KUKA KRL program: f1_Kuka_APT209T02S09.SRC

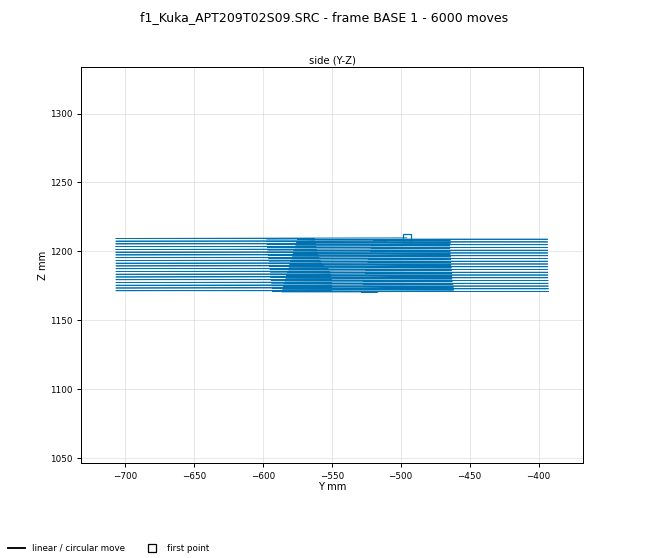
[picture p0: tool path of f1_Kuka_APT209T02S09.SRC in frame BASE 1, 6000 of 6001 moves have a stored position in this frame; points joined in program order, loops and branches not executed]
&ACCESS RVP
&REL 2
&PARAM TEMPLATE = C:\KRC\Roboter\Template\vorgabe
&PARAM EDITMASK = *
DEF f1_Kuka_APT209T02S09()


;FOLD INI;%{PE}%V3.2.0,%MKUKATPBASIS,%CINIT,%VCOMMON,%P
  ;FOLD BAS INI;%{E}%V3.2.0,%MKUKATPBASIS,%CINIT,%VINIT,%P
    GLOBAL INTERRUPT DECL 3 WHEN $STOPMESS==TRUE DO IR_STOPM ( )
    INTERRUPT ON 3
    BAS (#INITMOV,0 )
  ;ENDFOLD (BAS INI)
  ;FOLD USER INI;%{E}%V3.2.0,%MKUKATPUSER,%CINIT,%VINIT,%P
    ;Make your modifications here
  ;ENDFOLD (USER INI)
;ENDFOLD (INI)


;*** Make Null PTP Move
  PTP $pos_act

;*** Auto Load The Correct TOOL Data
  $tool=tool_data[2]

;*** Auto Load The Correct BASE Data
  $base=base_data[1]

  $ADVANCE = 5

;*** Restate Last Velocity
MMPM(30000.0)
SetRPM(8000)
LIN {X 0.139,Y -495.504,Z 1209.880,A 0.000,B 0.000,C 90.000,E1 194.426} C_DIS
LIN {X -0.101,Y -498.909,Z 1209.874,A 0.000,B 0.000,C 90.000,E1 193.244} C_DIS
LIN {X -0.001,Y -505.040,Z 1209.862,A 0.000,B 0.000,C 90.000,E1 191.130} C_DIS
LIN {X 0.236,Y -509.405,Z 1209.854,A 0.000,B 0.000,C 90.000,E1 189.613} C_DIS
LIN {X -0.068,Y -515.059,Z 1209.844,A 0.000,B 0.000,C 90.000,E1 187.871} C_DIS
LIN {X 0.218,Y -518.809,Z 1209.837,A 0.000,B 0.000,C 90.000,E1 186.663} C_DIS
LIN {X 0.043,Y -523.311,Z 1209.829,A 0.000,B 0.000,C 90.000,E1 185.220} C_DIS
LIN {X -0.139,Y -528.677,Z 1209.819,A 0.000,B 0.000,C 90.000,E1 183.498} C_DIS
LIN {X -0.218,Y -533.146,Z 1209.811,A 0.000,B 0.000,C 90.000,E1 182.064} C_DIS
LIN {X -0.220,Y -537.647,Z 1209.803,A 0.000,B 0.000,C 90.000,E1 180.630} C_DIS
LIN {X -0.152,Y -542.076,Z 1209.796,A 0.000,B 0.000,C 90.000,E1 179.198} C_DIS
LIN {X -0.025,Y -545.583,Z 1209.789,A 0.000,B 0.000,C 90.000,E1 178.051} C_DIS
LIN {X 0.254,Y -550.664,Z 1209.780,A 0.000,B 0.000,C 90.000,E1 176.331} C_DIS
LIN {X 0.057,Y -554.716,Z 1209.772,A 0.000,B 0.000,C 90.000,E1 174.951} C_DIS
LIN {X -0.073,Y -558.723,Z 1209.764,A 0.000,B 0.000,C 90.000,E1 173.571} C_DIS
LIN {X 0.229,Y -564.136,Z 1209.754,A 0.000,B 0.000,C 90.000,E1 171.602} C_DIS
LIN {X -0.065,Y -568.767,Z 1209.744,A 0.000,B 0.000,C 90.000,E1 169.982} C_DIS
LIN {X -0.066,Y -573.325,Z 1209.735,A 0.000,B 0.000,C 90.000,E1 168.342} C_DIS
LIN {X 0.038,Y -577.922,Z 1209.726,A 0.000,B 0.000,C 90.000,E1 166.700} C_DIS
LIN {X -0.191,Y -582.656,Z 1209.717,A 0.000,B 0.000,C 90.000,E1 165.102} C_DIS
LIN {X 0.077,Y -588.302,Z 1209.707,A 0.000,B 0.000,C 90.000,E1 163.196} C_DIS
LIN {X 0.217,Y -593.215,Z 1209.698,A 0.000,B 0.000,C 90.000,E1 161.583} C_DIS
LIN {X 0.145,Y -601.075,Z 1209.685,A 0.000,B 0.000,C 90.000,E1 159.209} C_DIS
LIN {X -0.248,Y -607.551,Z 1209.674,A 0.000,B 0.000,C 90.000,E1 157.411} C_DIS
LIN {X 0.351,Y -612.972,Z 1209.666,A 0.000,B 0.000,C 90.000,E1 155.793} C_DIS
LIN {X -0.046,Y -617.299,Z 1209.659,A 0.000,B 0.000,C 90.000,E1 154.537} C_DIS
LIN {X -0.107,Y -621.487,Z 1209.651,A 0.000,B 0.000,C 90.000,E1 153.256} C_DIS
LIN {X -0.107,Y -624.711,Z 1209.646,A 0.000,B 0.000,C 90.000,E1 152.231} C_DIS
LIN {X -0.265,Y -630.161,Z 1209.636,A 0.000,B 0.000,C 90.000,E1 150.461} C_DIS
LIN {X -0.368,Y -633.922,Z 1209.629,A 0.000,B 0.000,C 90.000,E1 149.203} C_DIS
LIN {X 0.090,Y -636.876,Z 1209.623,A 0.000,B 0.000,C 90.000,E1 148.152} C_DIS
LIN {X -0.114,Y -640.335,Z 1209.616,A 0.000,B 0.000,C 90.000,E1 146.914} C_DIS
LIN {X 0.231,Y -642.880,Z 1209.611,A 0.000,B 0.000,C 90.000,E1 145.881} C_DIS
LIN {X 0.127,Y -645.937,Z 1209.604,A 0.000,B 0.000,C 90.000,E1 144.642} C_DIS
LIN {X -0.080,Y -648.713,Z 1209.597,A 0.000,B 0.000,C 90.000,E1 143.417} C_DIS
LIN {X -0.235,Y -651.341,Z 1209.590,A 0.000,B 0.000,C 90.000,E1 142.190} C_DIS
LIN {X 0.060,Y -653.919,Z 1209.583,A 0.000,B 0.000,C 90.000,E1 140.928} C_DIS
LIN {X -0.103,Y -657.497,Z 1209.573,A 0.000,B 0.000,C 90.000,E1 139.218} C_DIS
LIN {X 0.237,Y -661.234,Z 1209.564,A 0.000,B 0.000,C 90.000,E1 137.472} C_DIS
LIN {X -0.311,Y -664.353,Z 1209.556,A 0.000,B 0.000,C 90.000,E1 136.053} C_DIS
LIN {X -0.324,Y -669.340,Z 1209.544,A 0.000,B 0.000,C 90.000,E1 133.866} C_DIS
LIN {X -0.205,Y -673.548,Z 1209.534,A 0.000,B 0.000,C 90.000,E1 132.162} C_DIS
LIN {X -0.016,Y -677.073,Z 1209.526,A 0.000,B 0.000,C 90.000,E1 130.701} C_DIS
LIN {X 0.170,Y -679.469,Z 1209.521,A 0.000,B 0.000,C 90.000,E1 129.725} C_DIS
LIN {X 0.021,Y -683.002,Z 1209.513,A 0.000,B 0.000,C 90.000,E1 128.302} C_DIS
LIN {X -0.325,Y -687.178,Z 1209.504,A 0.000,B 0.000,C 90.000,E1 126.664} C_DIS
LIN {X -0.075,Y -688.967,Z 1209.500,A 0.000,B 0.000,C 90.000,E1 125.931} C_DIS
LIN {X 0.231,Y -692.270,Z 1209.492,A 0.000,B 0.000,C 90.000,E1 124.485} C_DIS
LIN {X -0.226,Y -694.400,Z 1209.486,A 0.000,B 0.000,C 90.000,E1 123.579} C_DIS
LIN {X -0.426,Y -696.993,Z 1209.480,A 0.000,B 0.000,C 90.000,E1 122.418} C_DIS
LIN {X 0.093,Y -698.481,Z 1209.476,A 0.000,B 0.000,C 90.000,E1 121.671} C_DIS
LIN {X -0.055,Y -700.752,Z 1209.469,A 0.000,B 0.000,C 90.000,E1 120.512} C_DIS
LIN {X 0.075,Y -702.947,Z 1209.463,A 0.000,B 0.000,C 90.000,E1 119.333} C_DIS
LIN {X -0.041,Y -704.508,Z 1209.458,A 0.000,B 0.000,C 90.000,E1 118.409} C_DIS
LIN {X -0.425,Y -705.192,Z 1209.455,A 0.000,B 0.000,C 90.000,E1 117.975} C_DIS
LIN {X -0.181,Y -705.879,Z 1209.451,A 0.000,B 0.000,C 90.000,E1 117.257} C_DIS
LIN {X 0.043,Y -706.510,Z 1209.446,A 0.000,B 0.000,C 90.000,E1 116.309} C_DIS
LIN {X 0.292,Y -706.772,Z 1209.442,A 0.000,B 0.000,C 90.000,E1 115.591} C_DIS
LIN {X -0.060,Y -706.742,Z 1209.440,A 0.000,B 0.000,C 90.000,E1 115.155} C_DIS
LIN {X -0.115,Y -706.152,Z 1209.436,A 0.000,B 0.000,C 90.000,E1 114.463} C_DIS
LIN {X -0.177,Y -705.283,Z 1209.433,A 0.000,B 0.000,C 90.000,E1 114.003} C_DIS
LIN {X -0.175,Y -704.420,Z 1209.432,A 0.000,B 0.000,C 90.000,E1 113.770} C_DIS
LIN {X 0.391,Y -702.162,Z 1209.429,A 0.000,B 0.000,C 90.000,E1 113.259} C_DIS
LIN {X -0.391,Y -701.273,Z 1209.429,A 0.000,B 0.000,C 90.000,E1 113.206} C_DIS
LIN {X -0.049,Y -698.541,Z 1209.427,A 0.000,B 0.000,C 90.000,E1 112.950} C_DIS
LIN {X -0.168,Y -694.330,Z 1209.426,A 0.000,B 0.000,C 90.000,E1 112.642} C_DIS
LIN {X 0.180,Y -692.034,Z 1209.425,A 0.000,B 0.000,C 90.000,E1 112.514} C_DIS
LIN {X -0.156,Y -687.353,Z 1209.424,A 0.000,B 0.000,C 90.000,E1 112.386} C_DIS
LIN {X -0.201,Y -685.168,Z 1209.424,A 0.000,B 0.000,C 90.000,E1 112.333} C_DIS
LIN {X 0.019,Y -676.728,Z 1209.424,A 0.000,B 0.000,C 90.000,E1 112.280} C_DIS
LIN {X -0.017,Y -610.154,Z 1209.424,A 0.000,B 0.000,C 90.000,E1 112.280} C_DIS
LIN {X -0.099,Y -607.762,Z 1209.423,A 0.000,B 0.000,C 90.000,E1 112.153} C_DIS
LIN {X 0.206,Y -603.602,Z 1209.422,A 0.000,B 0.000,C 90.000,E1 111.844} C_DIS
LIN {X -0.326,Y -599.261,Z 1209.420,A 0.000,B 0.000,C 90.000,E1 111.535} C_DIS
LIN {X -0.044,Y -596.935,Z 1209.418,A 0.000,B 0.000,C 90.000,E1 111.280} C_DIS
LIN {X -0.020,Y -595.513,Z 1209.418,A 0.000,B 0.000,C 90.000,E1 111.153} C_DIS
LIN {X -0.208,Y -594.337,Z 1209.417,A 0.000,B 0.000,C 90.000,E1 111.046} C_DIS
LIN {X -0.049,Y -592.336,Z 1209.416,A 0.000,B 0.000,C 90.000,E1 110.791} C_DIS
LIN {X -0.092,Y -592.311,Z 1209.416,A 0.000,B 0.000,C 90.000,E1 110.791} C_DIS
LIN {X 0.096,Y -591.736,Z 1209.414,A 0.000,B 0.000,C 90.000,E1 110.482} C_DIS
LIN {X -0.232,Y -592.138,Z 1209.412,A 0.000,B 0.000,C 90.000,E1 110.248} C_DIS
LIN {X -0.086,Y -596.332,Z 1209.405,A 0.000,B 0.000,C 90.000,E1 108.906} C_DIS
LIN {X -0.199,Y -597.165,Z 1209.404,A 0.000,B 0.000,C 90.000,E1 108.652} C_DIS
LIN {X -0.167,Y -602.046,Z 1209.393,A 0.000,B 0.000,C 90.000,E1 106.804} C_DIS
LIN {X 0.023,Y -603.299,Z 1209.390,A 0.000,B 0.000,C 90.000,E1 106.260} C_DIS
LIN {X 0.260,Y -605.497,Z 1209.385,A 0.000,B 0.000,C 90.000,E1 105.190} C_DIS
LIN {X -0.065,Y -606.611,Z 1209.379,A 0.000,B 0.000,C 90.000,E1 104.175} C_DIS
LIN {X -0.266,Y -606.970,Z 1209.374,A 0.000,B 0.000,C 90.000,E1 103.411} C_DIS
LIN {X -0.199,Y -606.754,Z 1209.371,A 0.000,B 0.000,C 90.000,E1 102.883} C_DIS
LIN {X 0.129,Y -606.556,Z 1209.370,A 0.000,B 0.000,C 90.000,E1 102.591} C_DIS
LIN {X 0.195,Y -605.757,Z 1209.367,A 0.000,B 0.000,C 90.000,E1 102.063} C_DIS
LIN {X 0.255,Y -604.578,Z 1209.364,A 0.000,B 0.000,C 90.000,E1 101.535} C_DIS
LIN {X 0.305,Y -602.971,Z 1209.361,A 0.000,B 0.000,C 90.000,E1 101.007} C_DIS
LIN {X -0.084,Y -601.975,Z 1209.360,A 0.000,B 0.000,C 90.000,E1 100.782} C_DIS
LIN {X -0.048,Y -599.580,Z 1209.357,A 0.000,B 0.000,C 90.000,E1 100.254} C_DIS
LIN {X -0.035,Y -596.738,Z 1209.354,A 0.000,B 0.000,C 90.000,E1 99.726} C_DIS
LIN {X 0.055,Y -594.326,Z 1209.352,A 0.000,B 0.000,C 90.000,E1 99.321} C_DIS
LIN {X -0.180,Y -589.543,Z 1209.348,A 0.000,B 0.000,C 90.000,E1 98.681} C_DIS
LIN {X 0.248,Y -585.132,Z 1209.345,A 0.000,B 0.000,C 90.000,E1 98.106} C_DIS
LIN {X -0.230,Y -581.136,Z 1209.343,A 0.000,B 0.000,C 90.000,E1 97.757} C_DIS
LIN {X 0.097,Y -578.320,Z 1209.342,A 0.000,B 0.000,C 90.000,E1 97.473} C_DIS
LIN {X 0.147,Y -572.423,Z 1209.339,A 0.000,B 0.000,C 90.000,E1 97.004} C_DIS
LIN {X -0.278,Y -569.383,Z 1209.338,A 0.000,B 0.000,C 90.000,E1 96.834} C_DIS
LIN {X -0.203,Y -568.061,Z 1209.337,A 0.000,B 0.000,C 90.000,E1 96.720} C_DIS
LIN {X -0.262,Y -564.683,Z 1209.335,A 0.000,B 0.000,C 90.000,E1 96.372} C_DIS
LIN {X 0.221,Y -564.184,Z 1209.335,A 0.000,B 0.000,C 90.000,E1 96.258} C_DIS
LIN {X 0.042,Y -563.353,Z 1209.334,A 0.000,B 0.000,C 90.000,E1 96.087} C_DIS
LIN {X 0.089,Y -563.274,Z 1209.333,A 0.000,B 0.000,C 90.000,E1 95.910} C_DIS
LIN {X 0.180,Y -562.863,Z 1209.331,A 0.000,B 0.000,C 90.000,E1 95.625} C_DIS
LIN {X -0.049,Y -562.866,Z 1209.327,A 0.000,B 0.000,C 90.000,E1 94.821} C_DIS
LIN {X -0.096,Y -564.202,Z 1209.313,A 0.000,B 0.000,C 90.000,E1 92.350} C_DIS
LIN {X -0.212,Y -565.047,Z 1209.307,A 0.000,B 0.000,C 90.000,E1 91.260} C_DIS
LIN {X -0.217,Y -566.044,Z 1209.299,A 0.000,B 0.000,C 90.000,E1 89.885} C_DIS
LIN {X 0.166,Y -567.706,Z 1209.287,A 0.000,B 0.000,C 90.000,E1 87.650} C_DIS
LIN {X -0.069,Y -569.116,Z 1209.276,A 0.000,B 0.000,C 90.000,E1 85.755} C_DIS
LIN {X 0.169,Y -570.459,Z 1209.267,A 0.000,B 0.000,C 90.000,E1 84.090} C_DIS
LIN {X -0.015,Y -571.749,Z 1209.258,A 0.000,B 0.000,C 90.000,E1 82.470} C_DIS
LIN {X 0.209,Y -572.803,Z 1209.251,A 0.000,B 0.000,C 90.000,E1 81.084} C_DIS
LIN {X 0.169,Y -573.886,Z 1209.242,A 0.000,B 0.000,C 90.000,E1 79.454} C_DIS
LIN {X 0.144,Y -574.948,Z 1209.233,A 0.000,B 0.000,C 90.000,E1 77.825} C_DIS
LIN {X -0.177,Y -575.786,Z 1209.223,A 0.000,B 0.000,C 90.000,E1 76.228} C_DIS
LIN {X -0.266,Y -576.758,Z 1209.213,A 0.000,B 0.000,C 90.000,E1 74.338} C_DIS
LIN {X 0.161,Y -577.655,Z 1209.204,A 0.000,B 0.000,C 90.000,E1 72.670} C_DIS
LIN {X 0.062,Y -578.729,Z 1209.193,A 0.000,B 0.000,C 90.000,E1 70.786} C_DIS
LIN {X -0.004,Y -580.016,Z 1209.183,A 0.000,B 0.000,C 90.000,E1 68.901} C_DIS
LIN {X 0.155,Y -581.553,Z 1209.172,A 0.000,B 0.000,C 90.000,E1 66.997} C_DIS
LIN {X -0.123,Y -583.097,Z 1209.163,A 0.000,B 0.000,C 90.000,E1 65.409} C_DIS
LIN {X -0.079,Y -585.043,Z 1209.151,A 0.000,B 0.000,C 90.000,E1 63.256} C_DIS
LIN {X -0.014,Y -586.685,Z 1209.142,A 0.000,B 0.000,C 90.000,E1 61.641} C_DIS
LIN {X -0.144,Y -588.289,Z 1209.134,A 0.000,B 0.000,C 90.000,E1 60.049} C_DIS
LIN {X 0.196,Y -589.370,Z 1209.128,A 0.000,B 0.000,C 90.000,E1 58.948} C_DIS
LIN {X -0.079,Y -590.733,Z 1209.119,A 0.000,B 0.000,C 90.000,E1 57.375} C_DIS
LIN {X 0.171,Y -591.978,Z 1209.110,A 0.000,B 0.000,C 90.000,E1 55.754} C_DIS
LIN {X -0.203,Y -593.254,Z 1209.101,A 0.000,B 0.000,C 90.000,E1 54.196} C_DIS
LIN {X 0.283,Y -594.420,Z 1209.092,A 0.000,B 0.000,C 90.000,E1 52.557} C_DIS
LIN {X -0.108,Y -594.844,Z 1209.089,A 0.000,B 0.000,C 90.000,E1 52.065} C_DIS
LIN {X 0.068,Y -596.010,Z 1209.079,A 0.000,B 0.000,C 90.000,E1 50.194} C_DIS
LIN {X 0.058,Y -596.520,Z 1209.073,A 0.000,B 0.000,C 90.000,E1 49.138} C_DIS
LIN {X 0.049,Y -597.057,Z 1209.064,A 0.000,B 0.000,C 90.000,E1 47.553} C_DIS
LIN {X 0.012,Y -597.327,Z 1209.058,A 0.000,B 0.000,C 90.000,E1 46.500} C_DIS
LIN {X 0.197,Y -597.520,Z 1209.051,A 0.000,B 0.000,C 90.000,E1 45.162} C_DIS
LIN {X -0.047,Y -597.259,Z 1209.044,A 0.000,B 0.000,C 90.000,E1 43.866} C_DIS
LIN {X -0.086,Y -596.897,Z 1209.038,A 0.000,B 0.000,C 90.000,E1 42.813} C_DIS
LIN {X -0.098,Y -596.277,Z 1209.032,A 0.000,B 0.000,C 90.000,E1 41.757} C_DIS
LIN {X 0.119,Y -595.801,Z 1209.028,A 0.000,B 0.000,C 90.000,E1 40.943} C_DIS
LIN {X -0.130,Y -594.866,Z 1209.020,A 0.000,B 0.000,C 90.000,E1 39.644} C_DIS
LIN {X 0.075,Y -594.188,Z 1209.016,A 0.000,B 0.000,C 90.000,E1 38.830} C_DIS
LIN {X 0.271,Y -593.372,Z 1209.011,A 0.000,B 0.000,C 90.000,E1 38.016} C_DIS
LIN {X -0.162,Y -592.237,Z 1209.005,A 0.000,B 0.000,C 90.000,E1 36.996} C_DIS
LIN {X 0.069,Y -590.336,Z 1208.998,A 0.000,B 0.000,C 90.000,E1 35.644} C_DIS
LIN {X -0.274,Y -588.357,Z 1208.992,A 0.000,B 0.000,C 90.000,E1 34.612} C_DIS
LIN {X -0.014,Y -586.602,Z 1208.988,A 0.000,B 0.000,C 90.000,E1 33.785} C_DIS
LIN {X 0.225,Y -584.637,Z 1208.983,A 0.000,B 0.000,C 90.000,E1 32.959} C_DIS
LIN {X -0.363,Y -582.233,Z 1208.979,A 0.000,B 0.000,C 90.000,E1 32.212} C_DIS
LIN {X -0.175,Y -579.536,Z 1208.974,A 0.000,B 0.000,C 90.000,E1 31.386} C_DIS
LIN {X 0.326,Y -577.503,Z 1208.971,A 0.000,B 0.000,C 90.000,E1 30.797} C_DIS
LIN {X 0.161,Y -574.088,Z 1208.967,A 0.000,B 0.000,C 90.000,E1 30.001} C_DIS
LIN {X -0.041,Y -570.260,Z 1208.962,A 0.000,B 0.000,C 90.000,E1 29.205} C_DIS
LIN {X 0.298,Y -566.674,Z 1208.958,A 0.000,B 0.000,C 90.000,E1 28.487} C_DIS
LIN {X -0.066,Y -563.567,Z 1208.955,A 0.000,B 0.000,C 90.000,E1 27.975} C_DIS
LIN {X 0.212,Y -559.450,Z 1208.952,A 0.000,B 0.000,C 90.000,E1 27.257} C_DIS
LIN {X 0.090,Y -554.201,Z 1208.947,A 0.000,B 0.000,C 90.000,E1 26.437} C_DIS
LIN {X 0.157,Y -548.224,Z 1208.942,A 0.000,B 0.000,C 90.000,E1 25.591} C_DIS
LIN {X 0.045,Y -542.810,Z 1208.938,A 0.000,B 0.000,C 90.000,E1 24.899} C_DIS
LIN {X -0.110,Y -537.075,Z 1208.934,A 0.000,B 0.000,C 90.000,E1 24.207} C_DIS
LIN {X 0.042,Y -529.607,Z 1208.930,A 0.000,B 0.000,C 90.000,E1 23.334} C_DIS
LIN {X -0.095,Y -523.144,Z 1208.926,A 0.000,B 0.000,C 90.000,E1 22.642} C_DIS
LIN {X -0.038,Y -512.535,Z 1208.920,A 0.000,B 0.000,C 90.000,E1 21.535} C_DIS
LIN {X 0.089,Y -502.840,Z 1208.914,A 0.000,B 0.000,C 90.000,E1 20.556} C_DIS
LIN {X 0.092,Y -493.072,Z 1208.909,A 0.000,B 0.000,C 90.000,E1 19.631} C_DIS
LIN {X -0.078,Y -484.282,Z 1208.905,A 0.000,B 0.000,C 90.000,E1 18.852} C_DIS
LIN {X -0.191,Y -473.999,Z 1208.900,A 0.000,B 0.000,C 90.000,E1 17.946} C_DIS
LIN {X -0.210,Y -459.021,Z 1208.892,A 0.000,B 0.000,C 90.000,E1 16.622} C_DIS
LIN {X 0.052,Y -437.190,Z 1208.881,A 0.000,B 0.000,C 90.000,E1 14.537} C_DIS
LIN {X 0.049,Y -421.688,Z 1208.872,A 0.000,B 0.000,C 90.000,E1 12.939} C_DIS
LIN {X 0.085,Y -404.925,Z 1208.861,A 0.000,B 0.000,C 90.000,E1 11.007} C_DIS
LIN {X 0.068,Y -397.362,Z 1208.856,A 0.000,B 0.000,C 90.000,E1 10.018} C_DIS
LIN {X 0.048,Y -395.305,Z 1208.854,A 0.000,B 0.000,C 90.000,E1 9.670} C_DIS
LIN {X -0.151,Y -393.958,Z 1208.852,A 0.000,B 0.000,C 90.000,E1 9.434} C_DIS
LIN {X -0.107,Y -393.353,Z 1208.851,A 0.000,B 0.000,C 90.000,E1 9.151} C_DIS
LIN {X -0.144,Y -393.341,Z 1208.851,A 0.000,B 0.000,C 90.000,E1 9.151} C_DIS
LIN {X -0.068,Y -393.829,Z 1208.849,A 0.000,B 0.000,C 90.000,E1 8.803} C_DIS
LIN {X -0.142,Y -396.754,Z 1208.845,A 0.000,B 0.000,C 90.000,E1 8.106} C_DIS
LIN {X -0.187,Y -397.947,Z 1208.844,A 0.000,B 0.000,C 90.000,E1 7.936} C_DIS
LIN {X -0.212,Y -400.655,Z 1208.842,A 0.000,B 0.000,C 90.000,E1 7.587} C_DIS
LIN {X 0.204,Y -402.237,Z 1208.841,A 0.000,B 0.000,C 90.000,E1 7.352} C_DIS
LIN {X 0.215,Y -407.342,Z 1208.839,A 0.000,B 0.000,C 90.000,E1 6.891} C_DIS
LIN {X 0.092,Y -426.083,Z 1208.830,A 0.000,B 0.000,C 90.000,E1 5.454} C_DIS
LIN {X 0.154,Y -438.832,Z 1208.825,A 0.000,B 0.000,C 90.000,E1 4.473} C_DIS
LIN {X 0.215,Y -454.780,Z 1208.818,A 0.000,B 0.000,C 90.000,E1 3.269} C_DIS
LIN {X 0.037,Y -464.247,Z 1208.814,A 0.000,B 0.000,C 90.000,E1 2.579} C_DIS
LIN {X -0.223,Y -473.438,Z 1208.810,A 0.000,B 0.000,C 90.000,E1 1.892} C_DIS
LIN {X 0.079,Y -479.294,Z 1208.808,A 0.000,B 0.000,C 90.000,E1 1.375} C_DIS
LIN {X 0.100,Y -485.204,Z 1208.805,A 0.000,B 0.000,C 90.000,E1 0.859} C_DIS
LIN {X -0.057,Y -490.896,Z 1208.802,A 0.000,B 0.000,C 90.000,E1 0.344} C_DIS
LIN {X -0.023,Y -497.632,Z 1208.798,A 0.000,B 0.000,C 90.000,E1 359.656} C_DIS
LIN {X -0.115,Y -505.401,Z 1208.793,A 0.000,B 0.000,C 90.000,E1 358.797} C_DIS
LIN {X -0.060,Y -511.385,Z 1208.789,A 0.000,B 0.000,C 90.000,E1 358.051} C_DIS
LIN {X -0.010,Y -517.010,Z 1208.785,A 0.000,B 0.000,C 90.000,E1 357.306} C_DIS
LIN {X -0.117,Y -521.216,Z 1208.782,A 0.000,B 0.000,C 90.000,E1 356.731} C_DIS
LIN {X 0.013,Y -526.004,Z 1208.778,A 0.000,B 0.000,C 90.000,E1 355.988} C_DIS
LIN {X 0.221,Y -530.323,Z 1208.774,A 0.000,B 0.000,C 90.000,E1 355.241} C_DIS
LIN {X 0.215,Y -533.527,Z 1208.771,A 0.000,B 0.000,C 90.000,E1 354.666} C_DIS
LIN {X 0.233,Y -536.478,Z 1208.767,A 0.000,B 0.000,C 90.000,E1 354.090} C_DIS
LIN {X -0.206,Y -540.361,Z 1208.763,A 0.000,B 0.000,C 90.000,E1 353.280} C_DIS
LIN {X 0.131,Y -543.384,Z 1208.759,A 0.000,B 0.000,C 90.000,E1 352.534} C_DIS
LIN {X -0.245,Y -546.623,Z 1208.754,A 0.000,B 0.000,C 90.000,E1 351.724} C_DIS
LIN {X 0.040,Y -549.539,Z 1208.749,A 0.000,B 0.000,C 90.000,E1 350.849} C_DIS
LIN {X -0.157,Y -552.960,Z 1208.743,A 0.000,B 0.000,C 90.000,E1 349.746} C_DIS
LIN {X -0.207,Y -556.077,Z 1208.737,A 0.000,B 0.000,C 90.000,E1 348.634} C_DIS
LIN {X -0.208,Y -558.908,Z 1208.731,A 0.000,B 0.000,C 90.000,E1 347.521} C_DIS
LIN {X 0.223,Y -560.866,Z 1208.726,A 0.000,B 0.000,C 90.000,E1 346.645} C_DIS
LIN {X -0.129,Y -563.293,Z 1208.720,A 0.000,B 0.000,C 90.000,E1 345.574} C_DIS
LIN {X 0.264,Y -566.109,Z 1208.712,A 0.000,B 0.000,C 90.000,E1 344.157} C_DIS
LIN {X -0.018,Y -568.156,Z 1208.706,A 0.000,B 0.000,C 90.000,E1 343.087} C_DIS
LIN {X -0.107,Y -570.038,Z 1208.700,A 0.000,B 0.000,C 90.000,E1 342.000} C_DIS
LIN {X 0.208,Y -571.336,Z 1208.695,A 0.000,B 0.000,C 90.000,E1 341.148} C_DIS
LIN {X 0.168,Y -572.775,Z 1208.689,A 0.000,B 0.000,C 90.000,E1 340.061} C_DIS
LIN {X -0.023,Y -573.704,Z 1208.685,A 0.000,B 0.000,C 90.000,E1 339.263} C_DIS
LIN {X 0.165,Y -574.623,Z 1208.679,A 0.000,B 0.000,C 90.000,E1 338.156} C_DIS
LIN {X -0.009,Y -574.953,Z 1208.674,A 0.000,B 0.000,C 90.000,E1 337.358} C_DIS
LIN {X 0.043,Y -575.052,Z 1208.670,A 0.000,B 0.000,C 90.000,E1 336.538} C_DIS
LIN {X 0.022,Y -575.001,Z 1208.667,A 0.000,B 0.000,C 90.000,E1 335.997} C_DIS
LIN {X -0.084,Y -574.305,Z 1208.661,A 0.000,B 0.000,C 90.000,E1 334.921} C_DIS
LIN {X 0.119,Y -573.741,Z 1208.658,A 0.000,B 0.000,C 90.000,E1 334.357} C_DIS
LIN {X -0.106,Y -572.527,Z 1208.653,A 0.000,B 0.000,C 90.000,E1 333.563} C_DIS
LIN {X -0.080,Y -570.852,Z 1208.649,A 0.000,B 0.000,C 90.000,E1 332.743} C_DIS
LIN {X 0.186,Y -568.925,Z 1208.644,A 0.000,B 0.000,C 90.000,E1 331.897} C_DIS
LIN {X -0.067,Y -566.664,Z 1208.639,A 0.000,B 0.000,C 90.000,E1 331.101} C_DIS
LIN {X 0.064,Y -564.846,Z 1208.636,A 0.000,B 0.000,C 90.000,E1 330.539} C_DIS
LIN {X -0.036,Y -562.668,Z 1208.633,A 0.000,B 0.000,C 90.000,E1 329.999} C_DIS
LIN {X -0.046,Y -560.751,Z 1208.631,A 0.000,B 0.000,C 90.000,E1 329.587} C_DIS
LIN {X 0.310,Y -557.934,Z 1208.628,A 0.000,B 0.000,C 90.000,E1 328.997} C_DIS
LIN {X 0.053,Y -553.811,Z 1208.624,A 0.000,B 0.000,C 90.000,E1 328.329} C_DIS
LIN {X -0.240,Y -549.077,Z 1208.620,A 0.000,B 0.000,C 90.000,E1 327.661} C_DIS
LIN {X 0.181,Y -544.010,Z 1208.616,A 0.000,B 0.000,C 90.000,E1 326.914} C_DIS
LIN {X -0.061,Y -539.580,Z 1208.613,A 0.000,B 0.000,C 90.000,E1 326.373} C_DIS
LIN {X -0.096,Y -531.519,Z 1208.608,A 0.000,B 0.000,C 90.000,E1 325.388} C_DIS
LIN {X -0.021,Y -520.912,Z 1208.601,A 0.000,B 0.000,C 90.000,E1 324.116} C_DIS
LIN {X -0.117,Y -516.729,Z 1208.597,A 0.000,B 0.000,C 90.000,E1 323.543} C_DIS
LIN {X 0.087,Y -513.641,Z 1208.595,A 0.000,B 0.000,C 90.000,E1 323.004} C_DIS
LIN {X -0.102,Y -511.670,Z 1208.592,A 0.000,B 0.000,C 90.000,E1 322.557} C_DIS
LIN {X -0.151,Y -510.098,Z 1208.588,A 0.000,B 0.000,C 90.000,E1 321.823} C_DIS
LIN {X -0.035,Y -509.952,Z 1208.587,A 0.000,B 0.000,C 90.000,E1 321.662} C_DIS
LIN {X -0.302,Y -509.720,Z 1208.582,A 0.000,B 0.000,C 90.000,E1 320.803} C_DIS
LIN {X 0.095,Y -511.153,Z 1208.566,A 0.000,B 0.000,C 90.000,E1 317.796} C_DIS
LIN {X -0.044,Y -512.545,Z 1208.552,A 0.000,B 0.000,C 90.000,E1 315.445} C_DIS
LIN {X 0.158,Y -513.347,Z 1208.544,A 0.000,B 0.000,C 90.000,E1 313.947} C_DIS
LIN {X -0.085,Y -514.300,Z 1208.534,A 0.000,B 0.000,C 90.000,E1 312.204} C_DIS
LIN {X -0.018,Y -515.416,Z 1208.523,A 0.000,B 0.000,C 90.000,E1 310.135} C_DIS
LIN {X -0.236,Y -515.885,Z 1208.518,A 0.000,B 0.000,C 90.000,E1 309.277} C_DIS
LIN {X -0.252,Y -516.543,Z 1208.510,A 0.000,B 0.000,C 90.000,E1 307.810} C_DIS
LIN {X -0.042,Y -517.483,Z 1208.497,A 0.000,B 0.000,C 90.000,E1 305.438} C_DIS
LIN {X -0.165,Y -518.057,Z 1208.490,A 0.000,B 0.000,C 90.000,E1 304.278} C_DIS
LIN {X -0.050,Y -518.642,Z 1208.482,A 0.000,B 0.000,C 90.000,E1 302.801} C_DIS
LIN {X 0.284,Y -519.085,Z 1208.476,A 0.000,B 0.000,C 90.000,E1 301.592} C_DIS
LIN {X -0.085,Y -519.379,Z 1208.469,A 0.000,B 0.000,C 90.000,E1 300.463} C_DIS
LIN {X 0.003,Y -519.581,Z 1208.463,A 0.000,B 0.000,C 90.000,E1 299.283} C_DIS
LIN {X -0.231,Y -519.780,Z 1208.455,A 0.000,B 0.000,C 90.000,E1 297.847} C_DIS
LIN {X -0.007,Y -519.934,Z 1208.447,A 0.000,B 0.000,C 90.000,E1 296.360} C_DIS
LIN {X -0.012,Y -519.978,Z 1208.438,A 0.000,B 0.000,C 90.000,E1 294.899} C_DIS
LIN {X 0.120,Y -519.968,Z 1208.429,A 0.000,B 0.000,C 90.000,E1 293.131} C_DIS
LIN {X 0.178,Y -520.072,Z 1208.421,A 0.000,B 0.000,C 90.000,E1 291.663} C_DIS
LIN {X -0.237,Y -519.849,Z 1208.412,A 0.000,B 0.000,C 90.000,E1 290.248} C_DIS
LIN {X 0.199,Y -519.590,Z 1208.407,A 0.000,B 0.000,C 90.000,E1 289.322} C_DIS
LIN {X 0.056,Y -518.752,Z 1208.398,A 0.000,B 0.000,C 90.000,E1 287.583} C_DIS
LIN {X -0.083,Y -517.928,Z 1208.390,A 0.000,B 0.000,C 90.000,E1 286.134} C_DIS
LIN {X -0.025,Y -517.001,Z 1208.381,A 0.000,B 0.000,C 90.000,E1 284.662} C_DIS
LIN {X 0.130,Y -515.843,Z 1208.372,A 0.000,B 0.000,C 90.000,E1 282.883} C_DIS
LIN {X 0.024,Y -514.725,Z 1208.362,A 0.000,B 0.000,C 90.000,E1 281.130} C_DIS
LIN {X -0.107,Y -513.684,Z 1208.352,A 0.000,B 0.000,C 90.000,E1 279.378} C_DIS
LIN {X 0.240,Y -513.119,Z 1208.347,A 0.000,B 0.000,C 90.000,E1 278.454} C_DIS
LIN {X -0.089,Y -512.088,Z 1208.337,A 0.000,B 0.000,C 90.000,E1 276.720} C_DIS
LIN {X -0.040,Y -510.884,Z 1208.326,A 0.000,B 0.000,C 90.000,E1 274.645} C_DIS
LIN {X 0.139,Y -510.108,Z 1208.319,A 0.000,B 0.000,C 90.000,E1 273.440} C_DIS
LIN {X 0.145,Y -509.099,Z 1208.309,A 0.000,B 0.000,C 90.000,E1 271.661} C_DIS
LIN {X 0.098,Y -508.243,Z 1208.299,A 0.000,B 0.000,C 90.000,E1 269.885} C_DIS
LIN {X 0.045,Y -507.205,Z 1208.290,A 0.000,B 0.000,C 90.000,E1 268.108} C_DIS
LIN {X -0.031,Y -506.059,Z 1208.280,A 0.000,B 0.000,C 90.000,E1 266.331} C_DIS
LIN {X 0.000,Y -505.009,Z 1208.271,A 0.000,B 0.000,C 90.000,E1 264.837} C_DIS
LIN {X 0.128,Y -504.044,Z 1208.265,A 0.000,B 0.000,C 90.000,E1 263.628} C_DIS
LIN {X 0.163,Y -502.576,Z 1208.256,A 0.000,B 0.000,C 90.000,E1 262.129} C_DIS
LIN {X 0.168,Y -501.075,Z 1208.246,A 0.000,B 0.000,C 90.000,E1 260.330} C_DIS
LIN {X 0.082,Y -499.156,Z 1208.233,A 0.000,B 0.000,C 90.000,E1 257.937} C_DIS
LIN {X 0.203,Y -497.722,Z 1208.223,A 0.000,B 0.000,C 90.000,E1 256.117} C_DIS
LIN {X -0.072,Y -496.418,Z 1208.213,A 0.000,B 0.000,C 90.000,E1 254.338} C_DIS
LIN {X -0.135,Y -495.381,Z 1208.205,A 0.000,B 0.000,C 90.000,E1 252.834} C_DIS
LIN {X -0.299,Y -494.925,Z 1208.200,A 0.000,B 0.000,C 90.000,E1 251.945} C_DIS
LIN {X -0.185,Y -493.831,Z 1208.189,A 0.000,B 0.000,C 90.000,E1 250.115} C_DIS
LIN {X -0.135,Y -492.766,Z 1208.181,A 0.000,B 0.000,C 90.000,E1 248.592} C_DIS
LIN {X 0.068,Y -491.537,Z 1208.173,A 0.000,B 0.000,C 90.000,E1 247.050} C_DIS
LIN {X -0.013,Y -490.038,Z 1208.164,A 0.000,B 0.000,C 90.000,E1 245.537} C_DIS
LIN {X -0.120,Y -488.434,Z 1208.156,A 0.000,B 0.000,C 90.000,E1 244.024} C_DIS
LIN {X -0.056,Y -487.078,Z 1208.149,A 0.000,B 0.000,C 90.000,E1 242.794} C_DIS
LIN {X 0.010,Y -484.163,Z 1208.135,A 0.000,B 0.000,C 90.000,E1 240.333} C_DIS
LIN {X 0.046,Y -482.275,Z 1208.127,A 0.000,B 0.000,C 90.000,E1 238.791} C_DIS
LIN {X 0.061,Y -479.615,Z 1208.115,A 0.000,B 0.000,C 90.000,E1 236.628} C_DIS
LIN {X -0.129,Y -477.773,Z 1208.106,A 0.000,B 0.000,C 90.000,E1 235.102} C_DIS
LIN {X -0.076,Y -476.025,Z 1208.097,A 0.000,B 0.000,C 90.000,E1 233.543} C_DIS
LIN {X 0.179,Y -473.558,Z 1208.085,A 0.000,B 0.000,C 90.000,E1 231.331} C_DIS
LIN {X 0.136,Y -471.540,Z 1208.075,A 0.000,B 0.000,C 90.000,E1 229.461} C_DIS
LIN {X -0.071,Y -469.891,Z 1208.066,A 0.000,B 0.000,C 90.000,E1 227.919} C_DIS
LIN {X -0.233,Y -467.916,Z 1208.056,A 0.000,B 0.000,C 90.000,E1 226.053} C_DIS
LIN {X 0.135,Y -466.543,Z 1208.047,A 0.000,B 0.000,C 90.000,E1 224.433} C_DIS
LIN {X -0.036,Y -464.877,Z 1208.035,A 0.000,B 0.000,C 90.000,E1 222.243} C_DIS
LIN {X -0.196,Y -464.033,Z 1208.014,A 0.000,B 0.000,C 90.000,E1 218.463} C_DIS
LIN {X 0.170,Y -464.634,Z 1208.000,A 0.000,B 0.000,C 90.000,E1 215.884} C_DIS
LIN {X -0.130,Y -465.308,Z 1207.987,A 0.000,B 0.000,C 90.000,E1 213.706} C_DIS
LIN {X 0.080,Y -468.131,Z 1207.968,A 0.000,B 0.000,C 90.000,E1 210.207} C_DIS
LIN {X 0.017,Y -471.209,Z 1207.952,A 0.000,B 0.000,C 90.000,E1 207.385} C_DIS
LIN {X -0.057,Y -473.503,Z 1207.942,A 0.000,B 0.000,C 90.000,E1 205.515} C_DIS
LIN {X 0.021,Y -478.364,Z 1207.923,A 0.000,B 0.000,C 90.000,E1 202.078} C_DIS
LIN {X 0.094,Y -486.292,Z 1207.900,A 0.000,B 0.000,C 90.000,E1 198.055} C_DIS
LIN {X -0.083,Y -494.672,Z 1207.882,A 0.000,B 0.000,C 90.000,E1 194.717} C_DIS
LIN {X 0.176,Y -498.908,Z 1207.873,A 0.000,B 0.000,C 90.000,E1 193.175} C_DIS
LIN {X 0.168,Y -505.081,Z 1207.862,A 0.000,B 0.000,C 90.000,E1 191.074} C_DIS
LIN {X -0.045,Y -508.622,Z 1207.855,A 0.000,B 0.000,C 90.000,E1 189.905} C_DIS
LIN {X 0.113,Y -515.205,Z 1207.844,A 0.000,B 0.000,C 90.000,E1 187.814} C_DIS
LIN {X -0.112,Y -518.973,Z 1207.837,A 0.000,B 0.000,C 90.000,E1 186.663} C_DIS
LIN {X -0.277,Y -522.635,Z 1207.830,A 0.000,B 0.000,C 90.000,E1 185.511} C_DIS
LIN {X 0.061,Y -528.944,Z 1207.819,A 0.000,B 0.000,C 90.000,E1 183.440} C_DIS
LIN {X -0.012,Y -533.438,Z 1207.811,A 0.000,B 0.000,C 90.000,E1 182.007} C_DIS
LIN {X -0.005,Y -537.974,Z 1207.803,A 0.000,B 0.000,C 90.000,E1 180.573} C_DIS
LIN {X 0.072,Y -542.429,Z 1207.795,A 0.000,B 0.000,C 90.000,E1 179.141} C_DIS
LIN {X 0.204,Y -545.965,Z 1207.789,A 0.000,B 0.000,C 90.000,E1 177.993} C_DIS
LIN {X -0.057,Y -551.114,Z 1207.780,A 0.000,B 0.000,C 90.000,E1 176.331} C_DIS
LIN {X -0.247,Y -555.217,Z 1207.772,A 0.000,B 0.000,C 90.000,E1 174.951} C_DIS
LIN {X 0.117,Y -558.534,Z 1207.766,A 0.000,B 0.000,C 90.000,E1 173.799} C_DIS
LIN {X -0.212,Y -564.035,Z 1207.755,A 0.000,B 0.000,C 90.000,E1 171.894} C_DIS
LIN {X 0.141,Y -568.750,Z 1207.746,A 0.000,B 0.000,C 90.000,E1 170.208} C_DIS
LIN {X 0.236,Y -574.142,Z 1207.735,A 0.000,B 0.000,C 90.000,E1 168.285} C_DIS
LIN {X 0.010,Y -579.610,Z 1207.724,A 0.000,B 0.000,C 90.000,E1 166.408} C_DIS
LIN {X -0.188,Y -584.420,Z 1207.716,A 0.000,B 0.000,C 90.000,E1 164.810} C_DIS
LIN {X 0.117,Y -590.112,Z 1207.705,A 0.000,B 0.000,C 90.000,E1 162.906} C_DIS
LIN {X 0.032,Y -594.250,Z 1207.698,A 0.000,B 0.000,C 90.000,E1 161.583} C_DIS
LIN {X 0.287,Y -601.166,Z 1207.686,A 0.000,B 0.000,C 90.000,E1 159.444} C_DIS
LIN {X -0.326,Y -607.520,Z 1207.676,A 0.000,B 0.000,C 90.000,E1 157.667} C_DIS
LIN {X 0.267,Y -612.882,Z 1207.667,A 0.000,B 0.000,C 90.000,E1 156.049} C_DIS
LIN {X -0.133,Y -617.185,Z 1207.660,A 0.000,B 0.000,C 90.000,E1 154.793} C_DIS
LIN {X -0.199,Y -621.312,Z 1207.653,A 0.000,B 0.000,C 90.000,E1 153.512} C_DIS
LIN {X -0.195,Y -625.288,Z 1207.646,A 0.000,B 0.000,C 90.000,E1 152.231} C_DIS
LIN {X 0.135,Y -627.606,Z 1207.641,A 0.000,B 0.000,C 90.000,E1 151.435} C_DIS
LIN {X 0.024,Y -632.169,Z 1207.633,A 0.000,B 0.000,C 90.000,E1 149.921} C_DIS
LIN {X -0.006,Y -636.574,Z 1207.625,A 0.000,B 0.000,C 90.000,E1 148.408} C_DIS
LIN {X -0.169,Y -640.654,Z 1207.616,A 0.000,B 0.000,C 90.000,E1 146.914} C_DIS
LIN {X -0.308,Y -643.783,Z 1207.609,A 0.000,B 0.000,C 90.000,E1 145.674} C_DIS
LIN {X -0.026,Y -646.670,Z 1207.602,A 0.000,B 0.000,C 90.000,E1 144.402} C_DIS
LIN {X -0.125,Y -648.859,Z 1207.597,A 0.000,B 0.000,C 90.000,E1 143.417} C_DIS
LIN {X -0.278,Y -651.435,Z 1207.590,A 0.000,B 0.000,C 90.000,E1 142.190} C_DIS
LIN {X 0.018,Y -653.985,Z 1207.583,A 0.000,B 0.000,C 90.000,E1 140.928} C_DIS
LIN {X -0.143,Y -657.561,Z 1207.573,A 0.000,B 0.000,C 90.000,E1 139.218} C_DIS
LIN {X 0.198,Y -661.272,Z 1207.564,A 0.000,B 0.000,C 90.000,E1 137.472} C_DIS
LIN {X -0.349,Y -664.393,Z 1207.556,A 0.000,B 0.000,C 90.000,E1 136.053} C_DIS
LIN {X -0.361,Y -669.353,Z 1207.544,A 0.000,B 0.000,C 90.000,E1 133.866} C_DIS
LIN {X -0.242,Y -673.537,Z 1207.534,A 0.000,B 0.000,C 90.000,E1 132.162} C_DIS
LIN {X -0.054,Y -677.059,Z 1207.526,A 0.000,B 0.000,C 90.000,E1 130.701} C_DIS
LIN {X 0.160,Y -680.063,Z 1207.520,A 0.000,B 0.000,C 90.000,E1 129.483} C_DIS
LIN {X -0.408,Y -683.582,Z 1207.511,A 0.000,B 0.000,C 90.000,E1 128.096} C_DIS
LIN {X -0.149,Y -688.383,Z 1207.501,A 0.000,B 0.000,C 90.000,E1 126.171} C_DIS
LIN {X -0.019,Y -691.713,Z 1207.493,A 0.000,B 0.000,C 90.000,E1 124.739} C_DIS
LIN {X -0.266,Y -694.406,Z 1207.486,A 0.000,B 0.000,C 90.000,E1 123.579} C_DIS
LIN {X 0.149,Y -697.506,Z 1207.479,A 0.000,B 0.000,C 90.000,E1 122.133} C_DIS
LIN {X -0.374,Y -699.860,Z 1207.472,A 0.000,B 0.000,C 90.000,E1 121.003} C_DIS
LIN {X 0.099,Y -702.077,Z 1207.466,A 0.000,B 0.000,C 90.000,E1 119.795} C_DIS
LIN {X 0.255,Y -704.148,Z 1207.459,A 0.000,B 0.000,C 90.000,E1 118.615} C_DIS
LIN {X 0.158,Y -705.194,Z 1207.455,A 0.000,B 0.000,C 90.000,E1 117.924} C_DIS
LIN {X -0.222,Y -705.903,Z 1207.451,A 0.000,B 0.000,C 90.000,E1 117.257} C_DIS
LIN {X 0.003,Y -706.539,Z 1207.446,A 0.000,B 0.000,C 90.000,E1 116.309} C_DIS
LIN {X 0.251,Y -706.796,Z 1207.442,A 0.000,B 0.000,C 90.000,E1 115.591} C_DIS
LIN {X -0.100,Y -706.752,Z 1207.440,A 0.000,B 0.000,C 90.000,E1 115.155} C_DIS
LIN {X -0.154,Y -706.463,Z 1207.437,A 0.000,B 0.000,C 90.000,E1 114.695} C_DIS
LIN {X -0.154,Y -706.197,Z 1207.436,A 0.000,B 0.000,C 90.000,E1 114.463} C_DIS
LIN {X -0.216,Y -705.308,Z 1207.433,A 0.000,B 0.000,C 90.000,E1 114.003} C_DIS
LIN {X -0.214,Y -704.454,Z 1207.432,A 0.000,B 0.000,C 90.000,E1 113.770} C_DIS
LIN {X 0.352,Y -702.209,Z 1207.429,A 0.000,B 0.000,C 90.000,E1 113.259} C_DIS
LIN {X 0.214,Y -701.317,Z 1207.429,A 0.000,B 0.000,C 90.000,E1 113.153} C_DIS
LIN {X -0.084,Y -698.573,Z 1207.427,A 0.000,B 0.000,C 90.000,E1 112.950} C_DIS
LIN {X -0.052,Y -694.550,Z 1207.426,A 0.000,B 0.000,C 90.000,E1 112.642} C_DIS
LIN {X 0.279,Y -692.368,Z 1207.425,A 0.000,B 0.000,C 90.000,E1 112.514} C_DIS
LIN {X -0.075,Y -687.606,Z 1207.424,A 0.000,B 0.000,C 90.000,E1 112.386} C_DIS
LIN {X -0.119,Y -685.590,Z 1207.424,A 0.000,B 0.000,C 90.000,E1 112.333} C_DIS
LIN {X -0.359,Y -683.939,Z 1207.424,A 0.000,B 0.000,C 90.000,E1 112.333} C_DIS
LIN {X 0.037,Y -677.464,Z 1207.424,A 0.000,B 0.000,C 90.000,E1 112.280} C_DIS
LIN {X -0.003,Y -609.739,Z 1207.424,A 0.000,B 0.000,C 90.000,E1 112.280} C_DIS
LIN {X 0.208,Y -608.656,Z 1207.424,A 0.000,B 0.000,C 90.000,E1 112.206} C_DIS
LIN {X -0.159,Y -602.737,Z 1207.421,A 0.000,B 0.000,C 90.000,E1 111.844} C_DIS
LIN {X -0.044,Y -596.150,Z 1207.418,A 0.000,B 0.000,C 90.000,E1 111.280} C_DIS
LIN {X 0.050,Y -594.806,Z 1207.418,A 0.000,B 0.000,C 90.000,E1 111.153} C_DIS
LIN {X -0.335,Y -592.187,Z 1207.416,A 0.000,B 0.000,C 90.000,E1 110.918} C_DIS
LIN {X 0.095,Y -590.147,Z 1207.415,A 0.000,B 0.000,C 90.000,E1 110.684} C_DIS
LIN {X -0.151,Y -589.540,Z 1207.414,A 0.000,B 0.000,C 90.000,E1 110.610} C_DIS
LIN {X -0.256,Y -590.004,Z 1207.412,A 0.000,B 0.000,C 90.000,E1 110.120} C_DIS
LIN {X 0.174,Y -590.636,Z 1207.410,A 0.000,B 0.000,C 90.000,E1 109.812} C_DIS
LIN {X 0.098,Y -594.571,Z 1207.403,A 0.000,B 0.000,C 90.000,E1 108.489} C_DIS
LIN {X 0.121,Y -596.638,Z 1207.398,A 0.000,B 0.000,C 90.000,E1 107.692} C_DIS
LIN {X 0.260,Y -599.269,Z 1207.393,A 0.000,B 0.000,C 90.000,E1 106.622} C_DIS
LIN {X 0.146,Y -600.909,Z 1207.388,A 0.000,B 0.000,C 90.000,E1 105.843} C_DIS
LIN {X 0.165,Y -601.852,Z 1207.385,A 0.000,B 0.000,C 90.000,E1 105.315} C_DIS
LIN {X -0.234,Y -602.417,Z 1207.382,A 0.000,B 0.000,C 90.000,E1 104.828} C_DIS
LIN {X 0.108,Y -602.887,Z 1207.378,A 0.000,B 0.000,C 90.000,E1 104.008} C_DIS
LIN {X 0.148,Y -603.072,Z 1207.375,A 0.000,B 0.000,C 90.000,E1 103.480} C_DIS
LIN {X 0.192,Y -602.804,Z 1207.372,A 0.000,B 0.000,C 90.000,E1 102.952} C_DIS
LIN {X 0.052,Y -602.504,Z 1207.371,A 0.000,B 0.000,C 90.000,E1 102.703} C_DIS
LIN {X -0.039,Y -601.629,Z 1207.368,A 0.000,B 0.000,C 90.000,E1 102.187} C_DIS
LIN {X -0.004,Y -600.402,Z 1207.365,A 0.000,B 0.000,C 90.000,E1 101.658} C_DIS
LIN {X 0.022,Y -598.649,Z 1207.362,A 0.000,B 0.000,C 90.000,E1 101.130} C_DIS
LIN {X -0.168,Y -595.802,Z 1207.358,A 0.000,B 0.000,C 90.000,E1 100.489} C_DIS
LIN {X 0.202,Y -592.326,Z 1207.355,A 0.000,B 0.000,C 90.000,E1 99.792} C_DIS
LIN {X 0.162,Y -588.836,Z 1207.352,A 0.000,B 0.000,C 90.000,E1 99.265} C_DIS
LIN {X 0.003,Y -584.779,Z 1207.349,A 0.000,B 0.000,C 90.000,E1 98.746} C_DIS
LIN {X -0.093,Y -580.183,Z 1207.346,A 0.000,B 0.000,C 90.000,E1 98.219} C_DIS
LIN {X -0.081,Y -574.604,Z 1207.343,A 0.000,B 0.000,C 90.000,E1 97.701} C_DIS
LIN {X -0.205,Y -568.695,Z 1207.340,A 0.000,B 0.000,C 90.000,E1 97.239} C_DIS
LIN {X 0.237,Y -564.097,Z 1207.338,A 0.000,B 0.000,C 90.000,E1 96.720} C_DIS
LIN {X 0.196,Y -564.089,Z 1207.338,A 0.000,B 0.000,C 90.000,E1 96.720} C_DIS
LIN {X 0.106,Y -563.805,Z 1207.336,A 0.000,B 0.000,C 90.000,E1 96.486} C_DIS
LIN {X 0.079,Y -562.695,Z 1207.334,A 0.000,B 0.000,C 90.000,E1 96.144} C_DIS
LIN {X -0.038,Y -562.514,Z 1207.334,A 0.000,B 0.000,C 90.000,E1 96.087} C_DIS
LIN {X 0.018,Y -562.425,Z 1207.330,A 0.000,B 0.000,C 90.000,E1 95.391} C_DIS
LIN {X 0.083,Y -564.142,Z 1207.313,A 0.000,B 0.000,C 90.000,E1 92.350} C_DIS
LIN {X -0.034,Y -564.973,Z 1207.307,A 0.000,B 0.000,C 90.000,E1 91.260} C_DIS
LIN {X -0.041,Y -565.969,Z 1207.299,A 0.000,B 0.000,C 90.000,E1 89.885} C_DIS
LIN {X -0.227,Y -567.618,Z 1207.287,A 0.000,B 0.000,C 90.000,E1 87.707} C_DIS
LIN {X 0.105,Y -569.033,Z 1207.276,A 0.000,B 0.000,C 90.000,E1 85.755} C_DIS
LIN {X -0.227,Y -570.356,Z 1207.267,A 0.000,B 0.000,C 90.000,E1 84.147} C_DIS
LIN {X 0.154,Y -571.629,Z 1207.258,A 0.000,B 0.000,C 90.000,E1 82.470} C_DIS
LIN {X -0.190,Y -572.657,Z 1207.251,A 0.000,B 0.000,C 90.000,E1 81.141} C_DIS
LIN {X -0.231,Y -573.732,Z 1207.242,A 0.000,B 0.000,C 90.000,E1 79.511} C_DIS
LIN {X -0.256,Y -574.790,Z 1207.233,A 0.000,B 0.000,C 90.000,E1 77.881} C_DIS
LIN {X -0.019,Y -575.627,Z 1207.224,A 0.000,B 0.000,C 90.000,E1 76.228} C_DIS
LIN {X -0.111,Y -576.588,Z 1207.213,A 0.000,B 0.000,C 90.000,E1 74.338} C_DIS
LIN {X -0.239,Y -577.487,Z 1207.204,A 0.000,B 0.000,C 90.000,E1 72.725} C_DIS
LIN {X 0.209,Y -578.549,Z 1207.193,A 0.000,B 0.000,C 90.000,E1 70.786} C_DIS
LIN {X -0.250,Y -579.657,Z 1207.184,A 0.000,B 0.000,C 90.000,E1 69.209} C_DIS
LIN {X -0.240,Y -581.399,Z 1207.172,A 0.000,B 0.000,C 90.000,E1 67.050} C_DIS
LIN {X -0.116,Y -583.173,Z 1207.162,A 0.000,B 0.000,C 90.000,E1 65.153} C_DIS
LIN {X 0.054,Y -584.901,Z 1207.151,A 0.000,B 0.000,C 90.000,E1 63.256} C_DIS
LIN {X 0.117,Y -586.549,Z 1207.143,A 0.000,B 0.000,C 90.000,E1 61.641} C_DIS
LIN {X -0.016,Y -588.134,Z 1207.134,A 0.000,B 0.000,C 90.000,E1 60.049} C_DIS
LIN {X -0.183,Y -589.204,Z 1207.128,A 0.000,B 0.000,C 90.000,E1 58.997} C_DIS
LIN {X 0.044,Y -590.547,Z 1207.119,A 0.000,B 0.000,C 90.000,E1 57.375} C_DIS
LIN {X -0.407,Y -591.580,Z 1207.111,A 0.000,B 0.000,C 90.000,E1 56.087} C_DIS
LIN {X -0.088,Y -593.067,Z 1207.101,A 0.000,B 0.000,C 90.000,E1 54.196} C_DIS
LIN {X -0.078,Y -594.220,Z 1207.092,A 0.000,B 0.000,C 90.000,E1 52.603} C_DIS
LIN {X 0.003,Y -594.653,Z 1207.089,A 0.000,B 0.000,C 90.000,E1 52.065} C_DIS
LIN {X 0.174,Y -595.804,Z 1207.079,A 0.000,B 0.000,C 90.000,E1 50.194} C_DIS
LIN {X 0.161,Y -596.333,Z 1207.073,A 0.000,B 0.000,C 90.000,E1 49.138} C_DIS
LIN {X 0.148,Y -596.848,Z 1207.064,A 0.000,B 0.000,C 90.000,E1 47.553} C_DIS
LIN {X 0.109,Y -597.110,Z 1207.058,A 0.000,B 0.000,C 90.000,E1 46.500} C_DIS
LIN {X 0.290,Y -597.295,Z 1207.051,A 0.000,B 0.000,C 90.000,E1 45.162} C_DIS
LIN {X 0.041,Y -597.040,Z 1207.044,A 0.000,B 0.000,C 90.000,E1 43.866} C_DIS
LIN {X 0.000,Y -596.680,Z 1207.038,A 0.000,B 0.000,C 90.000,E1 42.813} C_DIS
LIN {X -0.015,Y -596.074,Z 1207.032,A 0.000,B 0.000,C 90.000,E1 41.757} C_DIS
LIN {X -0.250,Y -595.581,Z 1207.028,A 0.000,B 0.000,C 90.000,E1 40.987} C_DIS
LIN {X -0.054,Y -594.617,Z 1207.020,A 0.000,B 0.000,C 90.000,E1 39.644} C_DIS
LIN {X 0.149,Y -593.927,Z 1207.016,A 0.000,B 0.000,C 90.000,E1 38.830} C_DIS
LIN {X -0.023,Y -593.110,Z 1207.011,A 0.000,B 0.000,C 90.000,E1 38.051} C_DIS
LIN {X -0.094,Y -591.946,Z 1207.005,A 0.000,B 0.000,C 90.000,E1 36.996} C_DIS
LIN {X 0.131,Y -590.022,Z 1206.998,A 0.000,B 0.000,C 90.000,E1 35.644} C_DIS
LIN {X -0.216,Y -588.037,Z 1206.992,A 0.000,B 0.000,C 90.000,E1 34.612} C_DIS
LIN {X 0.040,Y -586.278,Z 1206.988,A 0.000,B 0.000,C 90.000,E1 33.785} C_DIS
LIN {X 0.276,Y -584.292,Z 1206.983,A 0.000,B 0.000,C 90.000,E1 32.959} C_DIS
LIN {X -0.316,Y -581.882,Z 1206.979,A 0.000,B 0.000,C 90.000,E1 32.212} C_DIS
LIN {X -0.278,Y -578.207,Z 1206.973,A 0.000,B 0.000,C 90.000,E1 31.131} C_DIS
LIN {X 0.064,Y -574.849,Z 1206.968,A 0.000,B 0.000,C 90.000,E1 30.285} C_DIS
LIN {X -0.043,Y -571.772,Z 1206.965,A 0.000,B 0.000,C 90.000,E1 29.617} C_DIS
LIN {X -0.180,Y -568.383,Z 1206.961,A 0.000,B 0.000,C 90.000,E1 28.949} C_DIS
LIN {X 0.235,Y -565.433,Z 1206.958,A 0.000,B 0.000,C 90.000,E1 28.359} C_DIS
LIN {X -0.136,Y -562.264,Z 1206.955,A 0.000,B 0.000,C 90.000,E1 27.847} C_DIS
LIN {X 0.028,Y -557.247,Z 1206.950,A 0.000,B 0.000,C 90.000,E1 27.001} C_DIS
LIN {X 0.103,Y -553.691,Z 1206.947,A 0.000,B 0.000,C 90.000,E1 26.437} C_DIS
LIN {X 0.281,Y -548.704,Z 1206.943,A 0.000,B 0.000,C 90.000,E1 25.720} C_DIS
LIN {X 0.174,Y -543.340,Z 1206.939,A 0.000,B 0.000,C 90.000,E1 25.027} C_DIS
LIN {X 0.021,Y -537.737,Z 1206.935,A 0.000,B 0.000,C 90.000,E1 24.335} C_DIS
LIN {X 0.183,Y -529.193,Z 1206.930,A 0.000,B 0.000,C 90.000,E1 23.334} C_DIS
LIN {X 0.019,Y -522.665,Z 1206.926,A 0.000,B 0.000,C 90.000,E1 22.642} C_DIS
LIN {X 0.177,Y -513.458,Z 1206.921,A 0.000,B 0.000,C 90.000,E1 21.663} C_DIS
LIN {X -0.196,Y -502.426,Z 1206.914,A 0.000,B 0.000,C 90.000,E1 20.610} C_DIS
LIN {X 0.257,Y -492.650,Z 1206.909,A 0.000,B 0.000,C 90.000,E1 19.631} C_DIS
LIN {X 0.062,Y -482.373,Z 1206.904,A 0.000,B 0.000,C 90.000,E1 18.725} C_DIS
LIN {X -0.026,Y -473.543,Z 1206.900,A 0.000,B 0.000,C 90.000,E1 17.946} C_DIS
LIN {X -0.080,Y -457.175,Z 1206.892,A 0.000,B 0.000,C 90.000,E1 16.496} C_DIS
LIN {X 0.139,Y -433.816,Z 1206.879,A 0.000,B 0.000,C 90.000,E1 14.245} C_DIS
LIN {X 0.071,Y -421.180,Z 1206.872,A 0.000,B 0.000,C 90.000,E1 12.939} C_DIS
LIN {X 0.088,Y -404.525,Z 1206.861,A 0.000,B 0.000,C 90.000,E1 11.007} C_DIS
LIN {X 0.156,Y -399.314,Z 1206.857,A 0.000,B 0.000,C 90.000,E1 10.310} C_DIS
LIN {X 0.144,Y -396.747,Z 1206.855,A 0.000,B 0.000,C 90.000,E1 9.962} C_DIS
LIN {X 0.074,Y -393.997,Z 1206.853,A 0.000,B 0.000,C 90.000,E1 9.443} C_DIS
LIN {X -0.005,Y -393.346,Z 1206.851,A 0.000,B 0.000,C 90.000,E1 9.151} C_DIS
LIN {X -0.043,Y -393.350,Z 1206.851,A 0.000,B 0.000,C 90.000,E1 9.151} C_DIS
LIN {X -0.166,Y -393.796,Z 1206.849,A 0.000,B 0.000,C 90.000,E1 8.859} C_DIS
LIN {X 0.003,Y -394.020,Z 1206.849,A 0.000,B 0.000,C 90.000,E1 8.746} C_DIS
LIN {X -0.069,Y -396.994,Z 1206.845,A 0.000,B 0.000,C 90.000,E1 8.049} C_DIS
LIN {X 0.144,Y -401.104,Z 1206.842,A 0.000,B 0.000,C 90.000,E1 7.473} C_DIS
LIN {X -0.146,Y -404.941,Z 1206.839,A 0.000,B 0.000,C 90.000,E1 7.125} C_DIS
LIN {X -0.085,Y -415.530,Z 1206.835,A 0.000,B 0.000,C 90.000,E1 6.258} C_DIS
LIN {X 0.107,Y -426.491,Z 1206.830,A 0.000,B 0.000,C 90.000,E1 5.391} C_DIS
LIN {X 0.127,Y -439.281,Z 1206.825,A 0.000,B 0.000,C 90.000,E1 4.416} C_DIS
LIN {X -0.085,Y -453.456,Z 1206.819,A 0.000,B 0.000,C 90.000,E1 3.383} C_DIS
LIN {X 0.187,Y -464.502,Z 1206.814,A 0.000,B 0.000,C 90.000,E1 2.522} C_DIS
LIN {X -0.064,Y -473.706,Z 1206.810,A 0.000,B 0.000,C 90.000,E1 1.835} C_DIS
LIN {X -0.210,Y -479.528,Z 1206.807,A 0.000,B 0.000,C 90.000,E1 1.375} C_DIS
LIN {X -0.064,Y -485.292,Z 1206.805,A 0.000,B 0.000,C 90.000,E1 0.859} C_DIS
LIN {X -0.238,Y -491.073,Z 1206.802,A 0.000,B 0.000,C 90.000,E1 0.344} C_DIS
LIN {X -0.023,Y -497.632,Z 1206.798,A 0.000,B 0.000,C 90.000,E1 359.656} C_DIS
LIN {X 0.009,Y -505.351,Z 1206.793,A 0.000,B 0.000,C 90.000,E1 358.797} C_DIS
LIN {X 0.064,Y -511.377,Z 1206.789,A 0.000,B 0.000,C 90.000,E1 358.051} C_DIS
LIN {X 0.038,Y -515.906,Z 1206.786,A 0.000,B 0.000,C 90.000,E1 357.478} C_DIS
LIN {X 0.153,Y -521.211,Z 1206.782,A 0.000,B 0.000,C 90.000,E1 356.731} C_DIS
LIN {X -0.239,Y -526.049,Z 1206.778,A 0.000,B 0.000,C 90.000,E1 356.045} C_DIS
LIN {X -0.031,Y -530.429,Z 1206.774,A 0.000,B 0.000,C 90.000,E1 355.298} C_DIS
LIN {X -0.037,Y -533.669,Z 1206.771,A 0.000,B 0.000,C 90.000,E1 354.723} C_DIS
LIN {X -0.293,Y -537.277,Z 1206.767,A 0.000,B 0.000,C 90.000,E1 354.033} C_DIS
LIN {X 0.078,Y -541.754,Z 1206.761,A 0.000,B 0.000,C 90.000,E1 352.996} C_DIS
LIN {X -0.045,Y -544.722,Z 1206.757,A 0.000,B 0.000,C 90.000,E1 352.299} C_DIS
LIN {X 0.137,Y -547.876,Z 1206.753,A 0.000,B 0.000,C 90.000,E1 351.432} C_DIS
LIN {X -0.208,Y -549.803,Z 1206.749,A 0.000,B 0.000,C 90.000,E1 350.905} C_DIS
LIN {X 0.144,Y -553.222,Z 1206.743,A 0.000,B 0.000,C 90.000,E1 349.746} C_DIS
LIN {X 0.100,Y -556.379,Z 1206.737,A 0.000,B 0.000,C 90.000,E1 348.634} C_DIS
LIN {X -0.038,Y -558.550,Z 1206.732,A 0.000,B 0.000,C 90.000,E1 347.813} C_DIS
LIN {X -0.006,Y -561.180,Z 1206.726,A 0.000,B 0.000,C 90.000,E1 346.700} C_DIS
LIN {X 0.054,Y -563.608,Z 1206.720,A 0.000,B 0.000,C 90.000,E1 345.589} C_DIS
LIN {X 0.048,Y -566.454,Z 1206.712,A 0.000,B 0.000,C 90.000,E1 344.212} C_DIS
LIN {X -0.063,Y -568.989,Z 1206.705,A 0.000,B 0.000,C 90.000,E1 342.851} C_DIS
LIN {X 0.234,Y -570.420,Z 1206.700,A 0.000,B 0.000,C 90.000,E1 342.000} C_DIS
LIN {X 0.180,Y -572.147,Z 1206.694,A 0.000,B 0.000,C 90.000,E1 340.913} C_DIS
LIN {X 0.146,Y -573.563,Z 1206.688,A 0.000,B 0.000,C 90.000,E1 339.826} C_DIS
LIN {X -0.040,Y -574.456,Z 1206.683,A 0.000,B 0.000,C 90.000,E1 339.028} C_DIS
LIN {X 0.152,Y -575.314,Z 1206.677,A 0.000,B 0.000,C 90.000,E1 337.922} C_DIS
LIN {X 0.046,Y -575.612,Z 1206.671,A 0.000,B 0.000,C 90.000,E1 336.847} C_DIS
LIN {X -0.122,Y -575.620,Z 1206.667,A 0.000,B 0.000,C 90.000,E1 336.049} C_DIS
LIN {X -0.277,Y -575.581,Z 1206.665,A 0.000,B 0.000,C 90.000,E1 335.793} C_DIS
LIN {X -0.215,Y -575.017,Z 1206.661,A 0.000,B 0.000,C 90.000,E1 334.973} C_DIS
LIN {X -0.005,Y -574.489,Z 1206.658,A 0.000,B 0.000,C 90.000,E1 334.409} C_DIS
LIN {X 0.041,Y -573.330,Z 1206.653,A 0.000,B 0.000,C 90.000,E1 333.589} C_DIS
LIN {X -0.179,Y -571.751,Z 1206.649,A 0.000,B 0.000,C 90.000,E1 332.794} C_DIS
LIN {X -0.168,Y -569.855,Z 1206.644,A 0.000,B 0.000,C 90.000,E1 331.975} C_DIS
LIN {X 0.084,Y -567.648,Z 1206.640,A 0.000,B 0.000,C 90.000,E1 331.129} C_DIS
LIN {X 0.002,Y -565.856,Z 1206.637,A 0.000,B 0.000,C 90.000,E1 330.589} C_DIS
LIN {X -0.087,Y -563.832,Z 1206.634,A 0.000,B 0.000,C 90.000,E1 330.049} C_DIS
LIN {X 0.012,Y -561.277,Z 1206.630,A 0.000,B 0.000,C 90.000,E1 329.488} C_DIS
LIN {X -0.113,Y -558.469,Z 1206.627,A 0.000,B 0.000,C 90.000,E1 328.948} C_DIS
LIN {X -0.076,Y -554.291,Z 1206.624,A 0.000,B 0.000,C 90.000,E1 328.250} C_DIS
LIN {X 0.104,Y -549.516,Z 1206.620,A 0.000,B 0.000,C 90.000,E1 327.533} C_DIS
LIN {X -0.101,Y -545.465,Z 1206.617,A 0.000,B 0.000,C 90.000,E1 326.993} C_DIS
LIN {X -0.034,Y -541.070,Z 1206.614,A 0.000,B 0.000,C 90.000,E1 326.421} C_DIS
LIN {X 0.307,Y -532.996,Z 1206.608,A 0.000,B 0.000,C 90.000,E1 325.388} C_DIS
LIN {X -0.106,Y -522.448,Z 1206.601,A 0.000,B 0.000,C 90.000,E1 324.196} C_DIS
LIN {X 0.157,Y -518.370,Z 1206.598,A 0.000,B 0.000,C 90.000,E1 323.623} C_DIS
LIN {X 0.043,Y -514.534,Z 1206.595,A 0.000,B 0.000,C 90.000,E1 323.050} C_DIS
LIN {X -0.216,Y -512.590,Z 1206.592,A 0.000,B 0.000,C 90.000,E1 322.637} C_DIS
LIN {X -0.098,Y -512.045,Z 1206.592,A 0.000,B 0.000,C 90.000,E1 322.477} C_DIS
LIN {X 0.283,Y -510.566,Z 1206.588,A 0.000,B 0.000,C 90.000,E1 321.823} C_DIS
LIN {X 0.084,Y -510.364,Z 1206.587,A 0.000,B 0.000,C 90.000,E1 321.698} C_DIS
LIN {X -0.097,Y -510.070,Z 1206.583,A 0.000,B 0.000,C 90.000,E1 320.928} C_DIS
LIN {X 0.230,Y -511.524,Z 1206.565,A 0.000,B 0.000,C 90.000,E1 317.634} C_DIS
LIN {X 0.206,Y -512.751,Z 1206.553,A 0.000,B 0.000,C 90.000,E1 315.567} C_DIS
LIN {X 0.053,Y -513.598,Z 1206.545,A 0.000,B 0.000,C 90.000,E1 314.109} C_DIS
LIN {X 0.078,Y -514.704,Z 1206.534,A 0.000,B 0.000,C 90.000,E1 312.043} C_DIS
LIN {X -0.179,Y -515.846,Z 1206.522,A 0.000,B 0.000,C 90.000,E1 310.011} C_DIS
LIN {X -0.197,Y -516.626,Z 1206.514,A 0.000,B 0.000,C 90.000,E1 308.543} C_DIS
LIN {X -0.203,Y -517.201,Z 1206.506,A 0.000,B 0.000,C 90.000,E1 307.076} C_DIS
LIN {X 0.143,Y -518.280,Z 1206.493,A 0.000,B 0.000,C 90.000,E1 304.692} C_DIS
LIN {X -0.020,Y -518.929,Z 1206.485,A 0.000,B 0.000,C 90.000,E1 303.245} C_DIS
LIN {X -0.176,Y -519.513,Z 1206.477,A 0.000,B 0.000,C 90.000,E1 301.799} C_DIS
LIN {X 0.173,Y -519.825,Z 1206.470,A 0.000,B 0.000,C 90.000,E1 300.590} C_DIS
LIN {X -0.062,Y -520.092,Z 1206.462,A 0.000,B 0.000,C 90.000,E1 299.155} C_DIS
LIN {X -0.287,Y -520.274,Z 1206.454,A 0.000,B 0.000,C 90.000,E1 297.719} C_DIS
LIN {X -0.053,Y -520.426,Z 1206.446,A 0.000,B 0.000,C 90.000,E1 296.232} C_DIS
LIN {X -0.194,Y -520.478,Z 1206.439,A 0.000,B 0.000,C 90.000,E1 295.079} C_DIS
LIN {X 0.067,Y -520.446,Z 1206.431,A 0.000,B 0.000,C 90.000,E1 293.590} C_DIS
LIN {X 0.007,Y -520.563,Z 1206.421,A 0.000,B 0.000,C 90.000,E1 291.844} C_DIS
LIN {X 0.088,Y -520.456,Z 1206.413,A 0.000,B 0.000,C 90.000,E1 290.375} C_DIS
LIN {X 0.042,Y -520.213,Z 1206.408,A 0.000,B 0.000,C 90.000,E1 289.504} C_DIS
LIN {X 0.050,Y -519.270,Z 1206.397,A 0.000,B 0.000,C 90.000,E1 287.457} C_DIS
LIN {X -0.228,Y -518.437,Z 1206.389,A 0.000,B 0.000,C 90.000,E1 286.024} C_DIS
LIN {X -0.008,Y -517.697,Z 1206.382,A 0.000,B 0.000,C 90.000,E1 284.828} C_DIS
LIN {X 0.034,Y -516.489,Z 1206.373,A 0.000,B 0.000,C 90.000,E1 283.063} C_DIS
LIN {X 0.049,Y -515.434,Z 1206.363,A 0.000,B 0.000,C 90.000,E1 281.299} C_DIS
LIN {X -0.183,Y -514.170,Z 1206.351,A 0.000,B 0.000,C 90.000,E1 279.265} C_DIS
LIN {X 0.117,Y -513.270,Z 1206.343,A 0.000,B 0.000,C 90.000,E1 277.757} C_DIS
LIN {X -0.177,Y -512.398,Z 1206.335,A 0.000,B 0.000,C 90.000,E1 276.315} C_DIS
LIN {X -0.074,Y -511.406,Z 1206.325,A 0.000,B 0.000,C 90.000,E1 274.531} C_DIS
LIN {X -0.126,Y -510.124,Z 1206.314,A 0.000,B 0.000,C 90.000,E1 272.465} C_DIS
LIN {X -0.229,Y -509.124,Z 1206.302,A 0.000,B 0.000,C 90.000,E1 270.401} C_DIS
LIN {X -0.086,Y -508.465,Z 1206.296,A 0.000,B 0.000,C 90.000,E1 269.198} C_DIS
LIN {X 0.059,Y -507.793,Z 1206.289,A 0.000,B 0.000,C 90.000,E1 267.993} C_DIS
LIN {X -0.008,Y -506.594,Z 1206.279,A 0.000,B 0.000,C 90.000,E1 266.216} C_DIS
LIN {X 0.031,Y -505.533,Z 1206.271,A 0.000,B 0.000,C 90.000,E1 264.723} C_DIS
LIN {X -0.217,Y -504.787,Z 1206.266,A 0.000,B 0.000,C 90.000,E1 263.856} C_DIS
LIN {X -0.094,Y -503.649,Z 1206.259,A 0.000,B 0.000,C 90.000,E1 262.648} C_DIS
LIN {X -0.061,Y -502.050,Z 1206.249,A 0.000,B 0.000,C 90.000,E1 260.849} C_DIS
LIN {X 0.078,Y -501.062,Z 1206.243,A 0.000,B 0.000,C 90.000,E1 259.634} C_DIS
LIN {X 0.137,Y -499.733,Z 1206.233,A 0.000,B 0.000,C 90.000,E1 257.825} C_DIS
LIN {X -0.181,Y -498.038,Z 1206.221,A 0.000,B 0.000,C 90.000,E1 255.755} C_DIS
LIN {X 0.127,Y -496.915,Z 1206.212,A 0.000,B 0.000,C 90.000,E1 254.212} C_DIS
LIN {X 0.031,Y -496.035,Z 1206.206,A 0.000,B 0.000,C 90.000,E1 253.015} C_DIS
LIN {X -0.079,Y -495.414,Z 1206.199,A 0.000,B 0.000,C 90.000,E1 251.819} C_DIS
LIN {X -0.117,Y -494.220,Z 1206.189,A 0.000,B 0.000,C 90.000,E1 250.007} C_DIS
LIN {X 0.112,Y -493.103,Z 1206.181,A 0.000,B 0.000,C 90.000,E1 248.465} C_DIS
LIN {X -0.172,Y -492.078,Z 1206.174,A 0.000,B 0.000,C 90.000,E1 247.283} C_DIS
LIN {X 0.043,Y -490.282,Z 1206.164,A 0.000,B 0.000,C 90.000,E1 245.433} C_DIS
LIN {X 0.144,Y -488.721,Z 1206.155,A 0.000,B 0.000,C 90.000,E1 243.896} C_DIS
LIN {X -0.013,Y -487.293,Z 1206.148,A 0.000,B 0.000,C 90.000,E1 242.692} C_DIS
LIN {X 0.062,Y -485.079,Z 1206.138,A 0.000,B 0.000,C 90.000,E1 240.845} C_DIS
LIN {X 0.068,Y -483.629,Z 1206.131,A 0.000,B 0.000,C 90.000,E1 239.616} C_DIS
LIN {X 0.090,Y -481.711,Z 1206.123,A 0.000,B 0.000,C 90.000,E1 238.074} C_DIS
LIN {X 0.138,Y -479.451,Z 1206.112,A 0.000,B 0.000,C 90.000,E1 236.215} C_DIS
LIN {X -0.056,Y -477.648,Z 1206.104,A 0.000,B 0.000,C 90.000,E1 234.689} C_DIS
LIN {X -0.010,Y -475.829,Z 1206.095,A 0.000,B 0.000,C 90.000,E1 233.130} C_DIS
LIN {X -0.140,Y -473.372,Z 1206.083,A 0.000,B 0.000,C 90.000,E1 230.964} C_DIS
LIN {X -0.185,Y -471.355,Z 1206.073,A 0.000,B 0.000,C 90.000,E1 229.094} C_DIS
LIN {X 0.103,Y -468.942,Z 1206.060,A 0.000,B 0.000,C 90.000,E1 226.863} C_DIS
LIN {X 0.044,Y -466.542,Z 1206.047,A 0.000,B 0.000,C 90.000,E1 224.352} C_DIS
LIN {X -0.010,Y -464.536,Z 1206.031,A 0.000,B 0.000,C 90.000,E1 221.515} C_DIS
LIN {X -0.045,Y -463.968,Z 1206.015,A 0.000,B 0.000,C 90.000,E1 218.669} C_DIS
LIN {X -0.063,Y -464.492,Z 1206.001,A 0.000,B 0.000,C 90.000,E1 216.137} C_DIS
LIN {X 0.148,Y -465.208,Z 1205.987,A 0.000,B 0.000,C 90.000,E1 213.579} C_DIS
LIN {X -0.045,Y -468.014,Z 1205.967,A 0.000,B 0.000,C 90.000,E1 210.129} C_DIS
LIN {X 0.135,Y -470.731,Z 1205.953,A 0.000,B 0.000,C 90.000,E1 207.590} C_DIS
LIN {X -0.062,Y -472.226,Z 1205.946,A 0.000,B 0.000,C 90.000,E1 206.360} C_DIS
LIN {X 0.145,Y -474.095,Z 1205.938,A 0.000,B 0.000,C 90.000,E1 204.771} C_DIS
LIN {X 0.131,Y -477.793,Z 1205.924,A 0.000,B 0.000,C 90.000,E1 202.280} C_DIS
LIN {X -0.110,Y -484.897,Z 1205.903,A 0.000,B 0.000,C 90.000,E1 198.598} C_DIS
LIN {X -0.216,Y -493.144,Z 1205.885,A 0.000,B 0.000,C 90.000,E1 195.245} C_DIS
LIN {X -0.080,Y -498.196,Z 1205.875,A 0.000,B 0.000,C 90.000,E1 193.411} C_DIS
LIN {X -0.072,Y -505.276,Z 1205.861,A 0.000,B 0.000,C 90.000,E1 191.007} C_DIS
LIN {X -0.155,Y -513.622,Z 1205.846,A 0.000,B 0.000,C 90.000,E1 188.341} C_DIS
LIN {X 0.158,Y -518.390,Z 1205.838,A 0.000,B 0.000,C 90.000,E1 186.834} C_DIS
LIN {X -0.017,Y -522.067,Z 1205.832,A 0.000,B 0.000,C 90.000,E1 185.682} C_DIS
LIN {X -0.184,Y -526.614,Z 1205.823,A 0.000,B 0.000,C 90.000,E1 184.245} C_DIS
LIN {X 0.257,Y -531.232,Z 1205.815,A 0.000,B 0.000,C 90.000,E1 182.751} C_DIS
LIN {X 0.225,Y -537.595,Z 1205.804,A 0.000,B 0.000,C 90.000,E1 180.745} C_DIS
LIN {X -0.245,Y -542.093,Z 1205.796,A 0.000,B 0.000,C 90.000,E1 179.370} C_DIS
LIN {X -0.083,Y -546.521,Z 1205.789,A 0.000,B 0.000,C 90.000,E1 177.936} C_DIS
LIN {X 0.164,Y -550.860,Z 1205.781,A 0.000,B 0.000,C 90.000,E1 176.502} C_DIS
LIN {X -0.026,Y -555.073,Z 1205.773,A 0.000,B 0.000,C 90.000,E1 175.122} C_DIS
LIN {X -0.146,Y -559.243,Z 1205.765,A 0.000,B 0.000,C 90.000,E1 173.742} C_DIS
LIN {X 0.019,Y -564.061,Z 1205.756,A 0.000,B 0.000,C 90.000,E1 172.064} C_DIS
LIN {X -0.095,Y -569.627,Z 1205.745,A 0.000,B 0.000,C 90.000,E1 170.151} C_DIS
LIN {X -0.183,Y -574.323,Z 1205.736,A 0.000,B 0.000,C 90.000,E1 168.522} C_DIS
LIN {X 0.153,Y -579.819,Z 1205.726,A 0.000,B 0.000,C 90.000,E1 166.589} C_DIS
LIN {X -0.043,Y -584.705,Z 1205.717,A 0.000,B 0.000,C 90.000,E1 164.991} C_DIS
LIN {X -0.298,Y -590.396,Z 1205.706,A 0.000,B 0.000,C 90.000,E1 163.142} C_DIS
LIN {X 0.067,Y -595.377,Z 1205.697,A 0.000,B 0.000,C 90.000,E1 161.511} C_DIS
LIN {X 0.157,Y -602.289,Z 1205.686,A 0.000,B 0.000,C 90.000,E1 159.390} C_DIS
LIN {X 0.356,Y -608.542,Z 1205.675,A 0.000,B 0.000,C 90.000,E1 157.539} C_DIS
LIN {X 0.167,Y -613.843,Z 1205.667,A 0.000,B 0.000,C 90.000,E1 155.997} C_DIS
LIN {X 0.040,Y -618.068,Z 1205.660,A 0.000,B 0.000,C 90.000,E1 154.717} C_DIS
LIN {X 0.000,Y -621.299,Z 1205.654,A 0.000,B 0.000,C 90.000,E1 153.691} C_DIS
LIN {X 0.011,Y -625.240,Z 1205.647,A 0.000,B 0.000,C 90.000,E1 152.410} C_DIS
LIN {X 0.062,Y -628.318,Z 1205.641,A 0.000,B 0.000,C 90.000,E1 151.385} C_DIS
LIN {X -0.044,Y -632.788,Z 1205.633,A 0.000,B 0.000,C 90.000,E1 149.871} C_DIS
LIN {X -0.106,Y -636.414,Z 1205.626,A 0.000,B 0.000,C 90.000,E1 148.614} C_DIS
LIN {X 0.116,Y -641.083,Z 1205.616,A 0.000,B 0.000,C 90.000,E1 146.834} C_DIS
LIN {X -0.010,Y -644.157,Z 1205.609,A 0.000,B 0.000,C 90.000,E1 145.595} C_DIS
LIN {X -0.194,Y -647.520,Z 1205.601,A 0.000,B 0.000,C 90.000,E1 144.116} C_DIS
LIN {X 0.191,Y -649.106,Z 1205.596,A 0.000,B 0.000,C 90.000,E1 143.336} C_DIS
LIN {X 0.047,Y -651.623,Z 1205.590,A 0.000,B 0.000,C 90.000,E1 142.110} C_DIS
LIN {X -0.063,Y -654.143,Z 1205.583,A 0.000,B 0.000,C 90.000,E1 140.884} C_DIS
LIN {X 0.196,Y -657.713,Z 1205.573,A 0.000,B 0.000,C 90.000,E1 139.138} C_DIS
LIN {X -0.391,Y -661.403,Z 1205.564,A 0.000,B 0.000,C 90.000,E1 137.472} C_DIS
LIN {X 0.012,Y -664.021,Z 1205.557,A 0.000,B 0.000,C 90.000,E1 136.215} C_DIS
LIN {X -0.010,Y -668.896,Z 1205.545,A 0.000,B 0.000,C 90.000,E1 134.028} C_DIS
LIN {X 0.101,Y -673.049,Z 1205.535,A 0.000,B 0.000,C 90.000,E1 132.324} C_DIS
LIN {X -0.248,Y -675.979,Z 1205.529,A 0.000,B 0.000,C 90.000,E1 131.148} C_DIS
LIN {X 0.093,Y -680.187,Z 1205.519,A 0.000,B 0.000,C 90.000,E1 129.439} C_DIS
LIN {X -0.041,Y -683.679,Z 1205.511,A 0.000,B 0.000,C 90.000,E1 128.016} C_DIS
LIN {X 0.218,Y -688.489,Z 1205.501,A 0.000,B 0.000,C 90.000,E1 126.091} C_DIS
LIN {X 0.112,Y -690.707,Z 1205.495,A 0.000,B 0.000,C 90.000,E1 125.152} C_DIS
LIN {X 0.454,Y -693.983,Z 1205.488,A 0.000,B 0.000,C 90.000,E1 123.706} C_DIS
LIN {X -0.102,Y -697.102,Z 1205.480,A 0.000,B 0.000,C 90.000,E1 122.339} C_DIS
LIN {X 0.330,Y -699.515,Z 1205.473,A 0.000,B 0.000,C 90.000,E1 121.131} C_DIS
LIN {X 0.110,Y -702.159,Z 1205.465,A 0.000,B 0.000,C 90.000,E1 119.745} C_DIS
LIN {X 0.275,Y -704.218,Z 1205.459,A 0.000,B 0.000,C 90.000,E1 118.565} C_DIS
LIN {X -0.111,Y -705.227,Z 1205.455,A 0.000,B 0.000,C 90.000,E1 117.897} C_DIS
LIN {X -0.194,Y -705.955,Z 1205.451,A 0.000,B 0.000,C 90.000,E1 117.206} C_DIS
LIN {X 0.351,Y -706.594,Z 1205.446,A 0.000,B 0.000,C 90.000,E1 116.232} C_DIS
LIN {X -0.346,Y -706.815,Z 1205.442,A 0.000,B 0.000,C 90.000,E1 115.591} C_DIS
LIN {X -0.403,Y -706.630,Z 1205.438,A 0.000,B 0.000,C 90.000,E1 114.899} C_DIS
LIN {X -0.110,Y -706.486,Z 1205.437,A 0.000,B 0.000,C 90.000,E1 114.643} C_DIS
LIN {X 0.183,Y -706.157,Z 1205.436,A 0.000,B 0.000,C 90.000,E1 114.387} C_DIS
LIN {X -0.169,Y -705.229,Z 1205.433,A 0.000,B 0.000,C 90.000,E1 113.951} C_DIS
LIN {X 0.121,Y -703.196,Z 1205.430,A 0.000,B 0.000,C 90.000,E1 113.462} C_DIS
LIN {X 0.262,Y -702.648,Z 1205.430,A 0.000,B 0.000,C 90.000,E1 113.334} C_DIS
LIN {X -0.243,Y -701.951,Z 1205.429,A 0.000,B 0.000,C 90.000,E1 113.259} C_DIS
LIN {X -0.106,Y -700.906,Z 1205.428,A 0.000,B 0.000,C 90.000,E1 113.131} C_DIS
LIN {X 0.024,Y -695.465,Z 1205.426,A 0.000,B 0.000,C 90.000,E1 112.695} C_DIS
LIN {X 0.132,Y -693.945,Z 1205.426,A 0.000,B 0.000,C 90.000,E1 112.589} C_DIS
LIN {X -0.086,Y -691.535,Z 1205.425,A 0.000,B 0.000,C 90.000,E1 112.514} C_DIS
LIN {X 0.299,Y -686.924,Z 1205.424,A 0.000,B 0.000,C 90.000,E1 112.333} C_DIS
LIN {X 0.265,Y -683.769,Z 1205.424,A 0.000,B 0.000,C 90.000,E1 112.280} C_DIS
LIN {X 0.039,Y -677.520,Z 1205.424,A 0.000,B 0.000,C 90.000,E1 112.280} C_DIS
LIN {X -0.024,Y -609.329,Z 1205.424,A 0.000,B 0.000,C 90.000,E1 112.280} C_DIS
LIN {X -0.061,Y -605.955,Z 1205.423,A 0.000,B 0.000,C 90.000,E1 112.078} C_DIS
LIN {X -0.241,Y -603.043,Z 1205.422,A 0.000,B 0.000,C 90.000,E1 111.897} C_DIS
LIN {X 0.136,Y -595.878,Z 1205.418,A 0.000,B 0.000,C 90.000,E1 111.280} C_DIS
LIN {X 0.190,Y -588.979,Z 1205.415,A 0.000,B 0.000,C 90.000,E1 110.663} C_DIS
LIN {X -0.034,Y -587.497,Z 1205.414,A 0.000,B 0.000,C 90.000,E1 110.482} C_DIS
LIN {X -0.077,Y -587.479,Z 1205.414,A 0.000,B 0.000,C 90.000,E1 110.482} C_DIS
LIN {X 0.275,Y -587.208,Z 1205.411,A 0.000,B 0.000,C 90.000,E1 109.993} C_DIS
LIN {X 0.128,Y -589.074,Z 1205.407,A 0.000,B 0.000,C 90.000,E1 109.322} C_DIS
LIN {X 0.226,Y -590.748,Z 1205.405,A 0.000,B 0.000,C 90.000,E1 108.779} C_DIS
LIN {X 0.023,Y -592.842,Z 1205.400,A 0.000,B 0.000,C 90.000,E1 108.000} C_DIS
LIN {X -0.017,Y -595.974,Z 1205.393,A 0.000,B 0.000,C 90.000,E1 106.677} C_DIS
LIN {X -0.167,Y -597.493,Z 1205.388,A 0.000,B 0.000,C 90.000,E1 105.898} C_DIS
LIN {X -0.174,Y -598.274,Z 1205.385,A 0.000,B 0.000,C 90.000,E1 105.371} C_DIS
LIN {X -0.017,Y -598.743,Z 1205.382,A 0.000,B 0.000,C 90.000,E1 104.828} C_DIS
LIN {X -0.296,Y -599.100,Z 1205.378,A 0.000,B 0.000,C 90.000,E1 104.064} C_DIS
LIN {X -0.283,Y -599.172,Z 1205.375,A 0.000,B 0.000,C 90.000,E1 103.536} C_DIS
LIN {X -0.268,Y -598.598,Z 1205.372,A 0.000,B 0.000,C 90.000,E1 103.008} C_DIS
LIN {X -0.254,Y -597.779,Z 1205.369,A 0.000,B 0.000,C 90.000,E1 102.479} C_DIS
LIN {X 0.043,Y -597.251,Z 1205.368,A 0.000,B 0.000,C 90.000,E1 102.187} C_DIS
LIN {X 0.048,Y -595.849,Z 1205.365,A 0.000,B 0.000,C 90.000,E1 101.658} C_DIS
LIN {X 0.043,Y -593.895,Z 1205.362,A 0.000,B 0.000,C 90.000,E1 101.130} C_DIS
LIN {X 0.022,Y -591.563,Z 1205.359,A 0.000,B 0.000,C 90.000,E1 100.602} C_DIS
LIN {X -0.230,Y -587.987,Z 1205.355,A 0.000,B 0.000,C 90.000,E1 99.962} C_DIS
LIN {X 0.277,Y -584.528,Z 1205.352,A 0.000,B 0.000,C 90.000,E1 99.378} C_DIS
LIN {X -0.128,Y -578.984,Z 1205.349,A 0.000,B 0.000,C 90.000,E1 98.746} C_DIS
LIN {X -0.127,Y -575.225,Z 1205.346,A 0.000,B 0.000,C 90.000,E1 98.341} C_DIS
LIN {X 0.102,Y -569.468,Z 1205.344,A 0.000,B 0.000,C 90.000,E1 97.814} C_DIS
LIN {X -0.111,Y -563.968,Z 1205.340,A 0.000,B 0.000,C 90.000,E1 97.239} C_DIS
LIN {X 0.044,Y -562.783,Z 1205.339,A 0.000,B 0.000,C 90.000,E1 97.004} C_DIS
LIN {X -0.197,Y -561.999,Z 1205.334,A 0.000,B 0.000,C 90.000,E1 96.201} C_DIS
LIN {X 0.270,Y -562.050,Z 1205.332,A 0.000,B 0.000,C 90.000,E1 95.739} C_DIS
LIN {X -0.068,Y -563.100,Z 1205.321,A 0.000,B 0.000,C 90.000,E1 93.841} C_DIS
LIN {X 0.011,Y -564.207,Z 1205.312,A 0.000,B 0.000,C 90.000,E1 92.178} C_DIS
LIN {X 0.005,Y -565.185,Z 1205.305,A 0.000,B 0.000,C 90.000,E1 90.802} C_DIS
LIN {X 0.005,Y -566.210,Z 1205.297,A 0.000,B 0.000,C 90.000,E1 89.427} C_DIS
LIN {X 0.272,Y -567.657,Z 1205.286,A 0.000,B 0.000,C 90.000,E1 87.478} C_DIS
LIN {X -0.085,Y -568.902,Z 1205.277,A 0.000,B 0.000,C 90.000,E1 85.869} C_DIS
LIN {X -0.243,Y -570.402,Z 1205.266,A 0.000,B 0.000,C 90.000,E1 83.970} C_DIS
LIN {X 0.075,Y -571.647,Z 1205.257,A 0.000,B 0.000,C 90.000,E1 82.299} C_DIS
LIN {X -0.276,Y -572.652,Z 1205.250,A 0.000,B 0.000,C 90.000,E1 80.971} C_DIS
LIN {X 0.238,Y -573.696,Z 1205.241,A 0.000,B 0.000,C 90.000,E1 79.285} C_DIS
LIN {X -0.240,Y -574.707,Z 1205.232,A 0.000,B 0.000,C 90.000,E1 77.701} C_DIS
LIN {X 0.001,Y -575.566,Z 1205.223,A 0.000,B 0.000,C 90.000,E1 76.047} C_DIS
LIN {X -0.089,Y -576.533,Z 1205.212,A 0.000,B 0.000,C 90.000,E1 74.157} C_DIS
LIN {X 0.137,Y -577.272,Z 1205.204,A 0.000,B 0.000,C 90.000,E1 72.779} C_DIS
LIN {X 0.204,Y -578.170,Z 1205.195,A 0.000,B 0.000,C 90.000,E1 71.148} C_DIS
LIN {X 0.129,Y -579.437,Z 1205.185,A 0.000,B 0.000,C 90.000,E1 69.263} C_DIS
LIN {X 0.002,Y -581.400,Z 1205.171,A 0.000,B 0.000,C 90.000,E1 66.847} C_DIS
LIN {X 0.023,Y -582.960,Z 1205.162,A 0.000,B 0.000,C 90.000,E1 65.229} C_DIS
LIN {X 0.056,Y -584.928,Z 1205.151,A 0.000,B 0.000,C 90.000,E1 63.076} C_DIS
LIN {X -0.284,Y -586.329,Z 1205.143,A 0.000,B 0.000,C 90.000,E1 61.769} C_DIS
LIN {X 0.089,Y -587.923,Z 1205.134,A 0.000,B 0.000,C 90.000,E1 60.127} C_DIS
LIN {X 0.101,Y -589.189,Z 1205.127,A 0.000,B 0.000,C 90.000,E1 58.791} C_DIS
LIN {X 0.010,Y -590.514,Z 1205.118,A 0.000,B 0.000,C 90.000,E1 57.199} C_DIS
LIN {X -0.121,Y -591.549,Z 1205.110,A 0.000,B 0.000,C 90.000,E1 55.881} C_DIS
LIN {X -0.019,Y -592.803,Z 1205.102,A 0.000,B 0.000,C 90.000,E1 54.276} C_DIS
LIN {X 0.236,Y -593.784,Z 1205.094,A 0.000,B 0.000,C 90.000,E1 52.924} C_DIS
LIN {X -0.186,Y -594.538,Z 1205.088,A 0.000,B 0.000,C 90.000,E1 51.904} C_DIS
LIN {X 0.224,Y -595.553,Z 1205.079,A 0.000,B 0.000,C 90.000,E1 50.275} C_DIS
LIN {X 0.206,Y -596.095,Z 1205.074,A 0.000,B 0.000,C 90.000,E1 49.218} C_DIS
LIN {X -0.030,Y -596.548,Z 1205.066,A 0.000,B 0.000,C 90.000,E1 47.919} C_DIS
LIN {X -0.267,Y -596.873,Z 1205.059,A 0.000,B 0.000,C 90.000,E1 46.620} C_DIS
LIN {X 0.320,Y -597.047,Z 1205.052,A 0.000,B 0.000,C 90.000,E1 45.243} C_DIS
LIN {X 0.288,Y -596.926,Z 1205.046,A 0.000,B 0.000,C 90.000,E1 44.190} C_DIS
LIN {X -0.160,Y -596.585,Z 1205.040,A 0.000,B 0.000,C 90.000,E1 43.176} C_DIS
LIN {X 0.008,Y -595.919,Z 1205.032,A 0.000,B 0.000,C 90.000,E1 41.838} C_DIS
LIN {X -0.239,Y -595.042,Z 1205.025,A 0.000,B 0.000,C 90.000,E1 40.539} C_DIS
LIN {X 0.187,Y -594.187,Z 1205.019,A 0.000,B 0.000,C 90.000,E1 39.439} C_DIS
LIN {X -0.075,Y -593.439,Z 1205.015,A 0.000,B 0.000,C 90.000,E1 38.669} C_DIS
LIN {X -0.036,Y -592.311,Z 1205.009,A 0.000,B 0.000,C 90.000,E1 37.604} C_DIS
LIN {X 0.136,Y -591.386,Z 1205.005,A 0.000,B 0.000,C 90.000,E1 36.790} C_DIS
LIN {X 0.011,Y -589.401,Z 1204.997,A 0.000,B 0.000,C 90.000,E1 35.471} C_DIS
LIN {X -0.002,Y -587.347,Z 1204.991,A 0.000,B 0.000,C 90.000,E1 34.405} C_DIS
LIN {X 0.246,Y -585.481,Z 1204.987,A 0.000,B 0.000,C 90.000,E1 33.579} C_DIS
LIN {X -0.018,Y -583.363,Z 1204.982,A 0.000,B 0.000,C 90.000,E1 32.801} C_DIS
LIN {X 0.013,Y -581.748,Z 1204.979,A 0.000,B 0.000,C 90.000,E1 32.260} C_DIS
LIN {X 0.033,Y -579.950,Z 1204.976,A 0.000,B 0.000,C 90.000,E1 31.720} C_DIS
LIN {X -0.110,Y -577.007,Z 1204.972,A 0.000,B 0.000,C 90.000,E1 30.924} C_DIS
LIN {X -0.279,Y -573.580,Z 1204.967,A 0.000,B 0.000,C 90.000,E1 30.129} C_DIS
LIN {X 0.263,Y -571.677,Z 1204.965,A 0.000,B 0.000,C 90.000,E1 29.667} C_DIS
LIN {X -0.072,Y -568.989,Z 1204.962,A 0.000,B 0.000,C 90.000,E1 29.155} C_DIS
LIN {X -0.147,Y -566.124,Z 1204.959,A 0.000,B 0.000,C 90.000,E1 28.615} C_DIS
LIN {X 0.248,Y -563.038,Z 1204.956,A 0.000,B 0.000,C 90.000,E1 28.025} C_DIS
LIN {X 0.057,Y -557.216,Z 1204.951,A 0.000,B 0.000,C 90.000,E1 27.078} C_DIS
LIN {X 0.271,Y -552.689,Z 1204.947,A 0.000,B 0.000,C 90.000,E1 26.360} C_DIS
LIN {X -0.180,Y -548.757,Z 1204.944,A 0.000,B 0.000,C 90.000,E1 25.848} C_DIS
LIN {X -0.282,Y -543.406,Z 1204.940,A 0.000,B 0.000,C 90.000,E1 25.155} C_DIS
LIN {X 0.284,Y -537.773,Z 1204.936,A 0.000,B 0.000,C 90.000,E1 24.387} C_DIS
LIN {X 0.071,Y -530.514,Z 1204.931,A 0.000,B 0.000,C 90.000,E1 23.567} C_DIS
LIN {X -0.212,Y -525.388,Z 1204.928,A 0.000,B 0.000,C 90.000,E1 23.025} C_DIS
LIN {X -0.100,Y -521.390,Z 1204.926,A 0.000,B 0.000,C 90.000,E1 22.589} C_DIS
LIN {X -0.177,Y -512.387,Z 1204.920,A 0.000,B 0.000,C 90.000,E1 21.663} C_DIS
LIN {X -0.118,Y -503.145,Z 1204.915,A 0.000,B 0.000,C 90.000,E1 20.737} C_DIS
LIN {X -0.134,Y -493.405,Z 1204.910,A 0.000,B 0.000,C 90.000,E1 19.812} C_DIS
LIN {X 0.096,Y -483.181,Z 1204.905,A 0.000,B 0.000,C 90.000,E1 18.852} C_DIS
LIN {X -0.134,Y -474.526,Z 1204.901,A 0.000,B 0.000,C 90.000,E1 18.109} C_DIS
LIN {X -0.141,Y -460.425,Z 1204.894,A 0.000,B 0.000,C 90.000,E1 16.858} C_DIS
LIN {X 0.035,Y -434.171,Z 1204.880,A 0.000,B 0.000,C 90.000,E1 14.356} C_DIS
LIN {X 0.092,Y -420.156,Z 1204.872,A 0.000,B 0.000,C 90.000,E1 12.883} C_DIS
LIN {X 0.064,Y -405.040,Z 1204.862,A 0.000,B 0.000,C 90.000,E1 11.130} C_DIS
LIN {X -0.129,Y -401.088,Z 1204.859,A 0.000,B 0.000,C 90.000,E1 10.658} C_DIS
LIN {X 0.096,Y -395.806,Z 1204.855,A 0.000,B 0.000,C 90.000,E1 9.849} C_DIS
LIN {X 0.157,Y -393.871,Z 1204.853,A 0.000,B 0.000,C 90.000,E1 9.443} C_DIS
LIN {X 0.039,Y -393.350,Z 1204.851,A 0.000,B 0.000,C 90.000,E1 9.151} C_DIS
LIN {X 0.000,Y -393.342,Z 1204.851,A 0.000,B 0.000,C 90.000,E1 9.151} C_DIS
LIN {X 0.000,Y -393.873,Z 1204.849,A 0.000,B 0.000,C 90.000,E1 8.803} C_DIS
LIN {X -0.073,Y -396.716,Z 1204.845,A 0.000,B 0.000,C 90.000,E1 8.106} C_DIS
LIN {X -0.117,Y -397.846,Z 1204.844,A 0.000,B 0.000,C 90.000,E1 7.936} C_DIS
LIN {X -0.073,Y -401.878,Z 1204.841,A 0.000,B 0.000,C 90.000,E1 7.409} C_DIS
LIN {X 0.052,Y -404.952,Z 1204.839,A 0.000,B 0.000,C 90.000,E1 7.068} C_DIS
LIN {X 0.078,Y -412.707,Z 1204.836,A 0.000,B 0.000,C 90.000,E1 6.429} C_DIS
LIN {X 0.038,Y -426.960,Z 1204.830,A 0.000,B 0.000,C 90.000,E1 5.334} C_DIS
LIN {X 0.168,Y -441.148,Z 1204.824,A 0.000,B 0.000,C 90.000,E1 4.245} C_DIS
LIN {X -0.106,Y -455.461,Z 1204.818,A 0.000,B 0.000,C 90.000,E1 3.212} C_DIS
LIN {X 0.204,Y -466.463,Z 1204.813,A 0.000,B 0.000,C 90.000,E1 2.350} C_DIS
LIN {X -0.102,Y -475.731,Z 1204.809,A 0.000,B 0.000,C 90.000,E1 1.661} C_DIS
LIN {X -0.021,Y -483.174,Z 1204.806,A 0.000,B 0.000,C 90.000,E1 1.031} C_DIS
LIN {X -0.096,Y -491.440,Z 1204.802,A 0.000,B 0.000,C 90.000,E1 0.286} C_DIS
LIN {X -0.027,Y -497.636,Z 1204.798,A 0.000,B 0.000,C 90.000,E1 359.656} C_DIS
LIN {X 0.072,Y -505.356,Z 1204.793,A 0.000,B 0.000,C 90.000,E1 358.797} C_DIS
LIN {X 0.130,Y -511.418,Z 1204.789,A 0.000,B 0.000,C 90.000,E1 358.051} C_DIS
LIN {X -0.040,Y -516.132,Z 1204.786,A 0.000,B 0.000,C 90.000,E1 357.478} C_DIS
LIN {X 0.078,Y -521.462,Z 1204.782,A 0.000,B 0.000,C 90.000,E1 356.731} C_DIS
LIN {X 0.211,Y -526.328,Z 1204.778,A 0.000,B 0.000,C 90.000,E1 355.988} C_DIS
LIN {X -0.104,Y -530.736,Z 1204.774,A 0.000,B 0.000,C 90.000,E1 355.298} C_DIS
LIN {X -0.108,Y -534.001,Z 1204.771,A 0.000,B 0.000,C 90.000,E1 354.723} C_DIS
LIN {X -0.088,Y -536.955,Z 1204.767,A 0.000,B 0.000,C 90.000,E1 354.147} C_DIS
LIN {X -0.189,Y -542.724,Z 1204.760,A 0.000,B 0.000,C 90.000,E1 352.875} C_DIS
LIN {X -0.024,Y -546.161,Z 1204.756,A 0.000,B 0.000,C 90.000,E1 352.008} C_DIS
LIN {X 0.177,Y -549.217,Z 1204.751,A 0.000,B 0.000,C 90.000,E1 351.141} C_DIS
LIN {X -0.246,Y -551.031,Z 1204.748,A 0.000,B 0.000,C 90.000,E1 350.622} C_DIS
LIN {X 0.214,Y -554.401,Z 1204.742,A 0.000,B 0.000,C 90.000,E1 349.454} C_DIS
LIN {X 0.188,Y -557.514,Z 1204.735,A 0.000,B 0.000,C 90.000,E1 348.342} C_DIS
LIN {X 0.063,Y -559.600,Z 1204.731,A 0.000,B 0.000,C 90.000,E1 347.521} C_DIS
LIN {X -0.286,Y -562.815,Z 1204.723,A 0.000,B 0.000,C 90.000,E1 346.172} C_DIS
LIN {X -0.067,Y -565.125,Z 1204.717,A 0.000,B 0.000,C 90.000,E1 345.046} C_DIS
LIN {X 0.186,Y -567.381,Z 1204.711,A 0.000,B 0.000,C 90.000,E1 343.921} C_DIS
LIN {X -0.122,Y -570.409,Z 1204.702,A 0.000,B 0.000,C 90.000,E1 342.308} C_DIS
LIN {X 0.173,Y -572.612,Z 1204.694,A 0.000,B 0.000,C 90.000,E1 340.913} C_DIS
LIN {X 0.144,Y -574.053,Z 1204.688,A 0.000,B 0.000,C 90.000,E1 339.826} C_DIS
LIN {X -0.037,Y -574.978,Z 1204.683,A 0.000,B 0.000,C 90.000,E1 339.028} C_DIS
LIN {X 0.164,Y -575.840,Z 1204.677,A 0.000,B 0.000,C 90.000,E1 337.922} C_DIS
LIN {X -0.155,Y -576.088,Z 1204.674,A 0.000,B 0.000,C 90.000,E1 337.411} C_DIS
LIN {X 0.057,Y -576.278,Z 1204.668,A 0.000,B 0.000,C 90.000,E1 336.305} C_DIS
LIN {X -0.250,Y -576.232,Z 1204.665,A 0.000,B 0.000,C 90.000,E1 335.793} C_DIS
LIN {X -0.181,Y -575.701,Z 1204.661,A 0.000,B 0.000,C 90.000,E1 334.973} C_DIS
LIN {X -0.118,Y -574.862,Z 1204.656,A 0.000,B 0.000,C 90.000,E1 334.152} C_DIS
LIN {X -0.070,Y -573.587,Z 1204.652,A 0.000,B 0.000,C 90.000,E1 333.332} C_DIS
LIN {X -0.125,Y -572.544,Z 1204.649,A 0.000,B 0.000,C 90.000,E1 332.794} C_DIS
LIN {X -0.106,Y -570.665,Z 1204.644,A 0.000,B 0.000,C 90.000,E1 331.975} C_DIS
LIN {X 0.155,Y -568.494,Z 1204.640,A 0.000,B 0.000,C 90.000,E1 331.129} C_DIS
LIN {X 0.078,Y -566.731,Z 1204.637,A 0.000,B 0.000,C 90.000,E1 330.589} C_DIS
LIN {X -0.102,Y -565.816,Z 1204.635,A 0.000,B 0.000,C 90.000,E1 330.333} C_DIS
LIN {X -0.192,Y -563.536,Z 1204.632,A 0.000,B 0.000,C 90.000,E1 329.793} C_DIS
LIN {X 0.287,Y -561.621,Z 1204.630,A 0.000,B 0.000,C 90.000,E1 329.331} C_DIS
LIN {X 0.168,Y -558.746,Z 1204.627,A 0.000,B 0.000,C 90.000,E1 328.791} C_DIS
LIN {X -0.080,Y -554.494,Z 1204.623,A 0.000,B 0.000,C 90.000,E1 328.122} C_DIS
LIN {X 0.097,Y -549.699,Z 1204.619,A 0.000,B 0.000,C 90.000,E1 327.406} C_DIS
LIN {X 0.191,Y -545.557,Z 1204.616,A 0.000,B 0.000,C 90.000,E1 326.834} C_DIS
LIN {X -0.040,Y -541.136,Z 1204.613,A 0.000,B 0.000,C 90.000,E1 326.294} C_DIS
LIN {X -0.289,Y -534.215,Z 1204.608,A 0.000,B 0.000,C 90.000,E1 325.468} C_DIS
LIN {X 0.227,Y -522.118,Z 1204.600,A 0.000,B 0.000,C 90.000,E1 323.989} C_DIS
LIN {X 0.125,Y -517.242,Z 1204.596,A 0.000,B 0.000,C 90.000,E1 323.336} C_DIS
LIN {X 0.031,Y -514.821,Z 1204.594,A 0.000,B 0.000,C 90.000,E1 322.970} C_DIS
LIN {X 0.222,Y -512.782,Z 1204.592,A 0.000,B 0.000,C 90.000,E1 322.477} C_DIS
LIN {X 0.029,Y -512.253,Z 1204.591,A 0.000,B 0.000,C 90.000,E1 322.351} C_DIS
LIN {X -0.190,Y -510.751,Z 1204.587,A 0.000,B 0.000,C 90.000,E1 321.743} C_DIS
LIN {X -0.166,Y -510.409,Z 1204.582,A 0.000,B 0.000,C 90.000,E1 320.723} C_DIS
LIN {X -0.119,Y -511.770,Z 1204.565,A 0.000,B 0.000,C 90.000,E1 317.757} C_DIS
LIN {X -0.273,Y -512.637,Z 1204.557,A 0.000,B 0.000,C 90.000,E1 316.296} C_DIS
LIN {X -0.169,Y -513.695,Z 1204.547,A 0.000,B 0.000,C 90.000,E1 314.514} C_DIS
LIN {X 0.152,Y -514.321,Z 1204.541,A 0.000,B 0.000,C 90.000,E1 313.299} C_DIS
LIN {X -0.035,Y -515.290,Z 1204.531,A 0.000,B 0.000,C 90.000,E1 311.553} C_DIS
LIN {X -0.193,Y -516.316,Z 1204.521,A 0.000,B 0.000,C 90.000,E1 309.806} C_DIS
LIN {X -0.134,Y -516.977,Z 1204.515,A 0.000,B 0.000,C 90.000,E1 308.624} C_DIS
LIN {X -0.131,Y -517.560,Z 1204.506,A 0.000,B 0.000,C 90.000,E1 307.156} C_DIS
LIN {X -0.195,Y -518.653,Z 1204.493,A 0.000,B 0.000,C 90.000,E1 304.818} C_DIS
LIN {X -0.356,Y -519.340,Z 1204.485,A 0.000,B 0.000,C 90.000,E1 303.372} C_DIS
LIN {X -0.130,Y -520.033,Z 1204.475,A 0.000,B 0.000,C 90.000,E1 301.592} C_DIS
LIN {X -0.037,Y -520.349,Z 1204.469,A 0.000,B 0.000,C 90.000,E1 300.413} C_DIS
LIN {X 0.326,Y -520.578,Z 1204.463,A 0.000,B 0.000,C 90.000,E1 299.205} C_DIS
LIN {X 0.104,Y -520.756,Z 1204.454,A 0.000,B 0.000,C 90.000,E1 297.769} C_DIS
LIN {X 0.109,Y -520.925,Z 1204.446,A 0.000,B 0.000,C 90.000,E1 296.309} C_DIS
LIN {X -0.020,Y -520.975,Z 1204.440,A 0.000,B 0.000,C 90.000,E1 295.155} C_DIS
LIN {X -0.011,Y -520.939,Z 1204.432,A 0.000,B 0.000,C 90.000,E1 293.695} C_DIS
LIN {X -0.072,Y -521.048,Z 1204.422,A 0.000,B 0.000,C 90.000,E1 291.950} C_DIS
LIN {X 0.007,Y -521.006,Z 1204.414,A 0.000,B 0.000,C 90.000,E1 290.482} C_DIS
LIN {X -0.212,Y -520.777,Z 1204.409,A 0.000,B 0.000,C 90.000,E1 289.631} C_DIS
LIN {X -0.166,Y -520.043,Z 1204.399,A 0.000,B 0.000,C 90.000,E1 287.873} C_DIS
LIN {X 0.066,Y -519.230,Z 1204.391,A 0.000,B 0.000,C 90.000,E1 286.386} C_DIS
LIN {X -0.199,Y -518.531,Z 1204.385,A 0.000,B 0.000,C 90.000,E1 285.245} C_DIS
LIN {X -0.029,Y -517.091,Z 1204.373,A 0.000,B 0.000,C 90.000,E1 283.175} C_DIS
LIN {X -0.109,Y -516.046,Z 1204.363,A 0.000,B 0.000,C 90.000,E1 281.422} C_DIS
LIN {X 0.278,Y -514.783,Z 1204.352,A 0.000,B 0.000,C 90.000,E1 279.321} C_DIS
LIN {X 0.130,Y -514.270,Z 1204.347,A 0.000,B 0.000,C 90.000,E1 278.454} C_DIS
LIN {X -0.174,Y -513.230,Z 1204.337,A 0.000,B 0.000,C 90.000,E1 276.720} C_DIS
LIN {X -0.095,Y -512.039,Z 1204.326,A 0.000,B 0.000,C 90.000,E1 274.645} C_DIS
LIN {X -0.132,Y -510.772,Z 1204.314,A 0.000,B 0.000,C 90.000,E1 272.579} C_DIS
LIN {X -0.219,Y -509.778,Z 1204.303,A 0.000,B 0.000,C 90.000,E1 270.516} C_DIS
LIN {X -0.156,Y -508.996,Z 1204.295,A 0.000,B 0.000,C 90.000,E1 269.026} C_DIS
LIN {X -0.004,Y -508.296,Z 1204.288,A 0.000,B 0.000,C 90.000,E1 267.822} C_DIS
LIN {X -0.063,Y -507.081,Z 1204.278,A 0.000,B 0.000,C 90.000,E1 266.045} C_DIS
LIN {X 0.030,Y -505.985,Z 1204.270,A 0.000,B 0.000,C 90.000,E1 264.546} C_DIS
LIN {X 0.239,Y -505.185,Z 1204.265,A 0.000,B 0.000,C 90.000,E1 263.628} C_DIS
LIN {X -0.203,Y -503.769,Z 1204.256,A 0.000,B 0.000,C 90.000,E1 262.186} C_DIS
LIN {X -0.167,Y -502.262,Z 1204.247,A 0.000,B 0.000,C 90.000,E1 260.387} C_DIS
LIN {X -0.214,Y -500.398,Z 1204.233,A 0.000,B 0.000,C 90.000,E1 257.993} C_DIS
LIN {X -0.097,Y -498.483,Z 1204.220,A 0.000,B 0.000,C 90.000,E1 255.574} C_DIS
LIN {X 0.131,Y -497.061,Z 1204.210,A 0.000,B 0.000,C 90.000,E1 253.740} C_DIS
LIN {X -0.020,Y -496.021,Z 1204.200,A 0.000,B 0.000,C 90.000,E1 251.945} C_DIS
LIN {X 0.118,Y -494.764,Z 1204.190,A 0.000,B 0.000,C 90.000,E1 250.115} C_DIS
LIN {X 0.044,Y -494.340,Z 1204.186,A 0.000,B 0.000,C 90.000,E1 249.518} C_DIS
LIN {X -0.182,Y -493.150,Z 1204.178,A 0.000,B 0.000,C 90.000,E1 248.028} C_DIS
LIN {X -0.011,Y -491.961,Z 1204.171,A 0.000,B 0.000,C 90.000,E1 246.794} C_DIS
LIN {X -0.079,Y -490.457,Z 1204.163,A 0.000,B 0.000,C 90.000,E1 245.281} C_DIS
LIN {X -0.177,Y -488.910,Z 1204.154,A 0.000,B 0.000,C 90.000,E1 243.768} C_DIS
LIN {X -0.105,Y -487.447,Z 1204.147,A 0.000,B 0.000,C 90.000,E1 242.538} C_DIS
LIN {X -0.057,Y -485.617,Z 1204.139,A 0.000,B 0.000,C 90.000,E1 241.001} C_DIS
LIN {X -0.020,Y -483.386,Z 1204.129,A 0.000,B 0.000,C 90.000,E1 239.154} C_DIS
LIN {X -0.199,Y -481.080,Z 1204.118,A 0.000,B 0.000,C 90.000,E1 237.327} C_DIS
LIN {X 0.031,Y -478.499,Z 1204.106,A 0.000,B 0.000,C 90.000,E1 235.135} C_DIS
LIN {X -0.117,Y -476.335,Z 1204.096,A 0.000,B 0.000,C 90.000,E1 233.290} C_DIS
LIN {X 0.058,Y -473.780,Z 1204.084,A 0.000,B 0.000,C 90.000,E1 231.090} C_DIS
LIN {X 0.027,Y -471.733,Z 1204.073,A 0.000,B 0.000,C 90.000,E1 229.218} C_DIS
LIN {X 0.016,Y -469.240,Z 1204.061,A 0.000,B 0.000,C 90.000,E1 227.025} C_DIS
LIN {X 0.035,Y -466.475,Z 1204.046,A 0.000,B 0.000,C 90.000,E1 224.190} C_DIS
LIN {X -0.024,Y -464.463,Z 1204.030,A 0.000,B 0.000,C 90.000,E1 221.353} C_DIS
LIN {X 0.009,Y -464.409,Z 1204.000,A 0.000,B 0.000,C 90.000,E1 215.964} C_DIS
LIN {X -0.293,Y -464.955,Z 1203.988,A 0.000,B 0.000,C 90.000,E1 213.785} C_DIS
LIN {X 0.140,Y -465.727,Z 1203.980,A 0.000,B 0.000,C 90.000,E1 212.467} C_DIS
LIN {X 0.060,Y -467.961,Z 1203.966,A 0.000,B 0.000,C 90.000,E1 209.951} C_DIS
LIN {X -0.004,Y -471.063,Z 1203.951,A 0.000,B 0.000,C 90.000,E1 207.129} C_DIS
LIN {X 0.060,Y -472.176,Z 1203.946,A 0.000,B 0.000,C 90.000,E1 206.181} C_DIS
LIN {X -0.179,Y -477.807,Z 1203.923,A 0.000,B 0.000,C 90.000,E1 202.153} C_DIS
LIN {X 0.030,Y -485.078,Z 1203.902,A 0.000,B 0.000,C 90.000,E1 198.417} C_DIS
LIN {X -0.068,Y -493.422,Z 1203.884,A 0.000,B 0.000,C 90.000,E1 195.064} C_DIS
LIN {X -0.011,Y -499.398,Z 1203.872,A 0.000,B 0.000,C 90.000,E1 192.939} C_DIS
LIN {X 0.051,Y -504.782,Z 1203.862,A 0.000,B 0.000,C 90.000,E1 191.130} C_DIS
LIN {X 0.045,Y -513.174,Z 1203.847,A 0.000,B 0.000,C 90.000,E1 188.454} C_DIS
LIN {X -0.142,Y -517.037,Z 1203.840,A 0.000,B 0.000,C 90.000,E1 187.296} C_DIS
LIN {X 0.178,Y -520.806,Z 1203.834,A 0.000,B 0.000,C 90.000,E1 186.087} C_DIS
LIN {X 0.037,Y -525.414,Z 1203.826,A 0.000,B 0.000,C 90.000,E1 184.645} C_DIS
LIN {X -0.103,Y -530.978,Z 1203.816,A 0.000,B 0.000,C 90.000,E1 182.922} C_DIS
LIN {X -0.147,Y -537.381,Z 1203.805,A 0.000,B 0.000,C 90.000,E1 180.917} C_DIS
LIN {X -0.083,Y -541.948,Z 1203.797,A 0.000,B 0.000,C 90.000,E1 179.484} C_DIS
LIN {X 0.079,Y -546.413,Z 1203.789,A 0.000,B 0.000,C 90.000,E1 178.051} C_DIS
LIN {X -0.222,Y -550.791,Z 1203.781,A 0.000,B 0.000,C 90.000,E1 176.674} C_DIS
LIN {X 0.093,Y -555.051,Z 1203.774,A 0.000,B 0.000,C 90.000,E1 175.241} C_DIS
LIN {X 0.024,Y -559.299,Z 1203.766,A 0.000,B 0.000,C 90.000,E1 173.856} C_DIS
LIN {X 0.274,Y -564.984,Z 1203.755,A 0.000,B 0.000,C 90.000,E1 171.894} C_DIS
LIN {X 0.177,Y -570.579,Z 1203.745,A 0.000,B 0.000,C 90.000,E1 169.982} C_DIS
LIN {X 0.015,Y -574.556,Z 1203.737,A 0.000,B 0.000,C 90.000,E1 168.634} C_DIS
LIN {X 0.149,Y -579.317,Z 1203.728,A 0.000,B 0.000,C 90.000,E1 166.992} C_DIS
LIN {X 0.140,Y -583.398,Z 1203.720,A 0.000,B 0.000,C 90.000,E1 165.644} C_DIS
LIN {X 0.177,Y -588.314,Z 1203.711,A 0.000,B 0.000,C 90.000,E1 164.031} C_DIS
LIN {X 0.017,Y -594.107,Z 1203.701,A 0.000,B 0.000,C 90.000,E1 162.181} C_DIS
LIN {X 0.163,Y -600.022,Z 1203.691,A 0.000,B 0.000,C 90.000,E1 160.315} C_DIS
LIN {X -0.125,Y -604.383,Z 1203.683,A 0.000,B 0.000,C 90.000,E1 159.028} C_DIS
LIN {X 0.167,Y -609.672,Z 1203.675,A 0.000,B 0.000,C 90.000,E1 157.433} C_DIS
LIN {X -0.292,Y -614.007,Z 1203.668,A 0.000,B 0.000,C 90.000,E1 156.177} C_DIS
LIN {X 0.144,Y -618.229,Z 1203.660,A 0.000,B 0.000,C 90.000,E1 154.845} C_DIS
LIN {X 0.103,Y -622.206,Z 1203.653,A 0.000,B 0.000,C 90.000,E1 153.563} C_DIS
LIN {X 0.130,Y -626.105,Z 1203.646,A 0.000,B 0.000,C 90.000,E1 152.281} C_DIS
LIN {X 0.173,Y -628.414,Z 1203.642,A 0.000,B 0.000,C 90.000,E1 151.513} C_DIS
LIN {X 0.071,Y -632.812,Z 1203.633,A 0.000,B 0.000,C 90.000,E1 149.999} C_DIS
LIN {X 0.012,Y -636.395,Z 1203.626,A 0.000,B 0.000,C 90.000,E1 148.742} C_DIS
LIN {X 0.342,Y -639.675,Z 1203.619,A 0.000,B 0.000,C 90.000,E1 147.454} C_DIS
LIN {X 0.283,Y -641.613,Z 1203.615,A 0.000,B 0.000,C 90.000,E1 146.707} C_DIS
LIN {X 0.115,Y -644.063,Z 1203.610,A 0.000,B 0.000,C 90.000,E1 145.722} C_DIS
LIN {X -0.013,Y -646.288,Z 1203.604,A 0.000,B 0.000,C 90.000,E1 144.736} C_DIS
LIN {X -0.064,Y -648.980,Z 1203.597,A 0.000,B 0.000,C 90.000,E1 143.497} C_DIS
LIN {X 0.158,Y -652.441,Z 1203.588,A 0.000,B 0.000,C 90.000,E1 141.743} C_DIS
LIN {X 0.008,Y -655.405,Z 1203.579,A 0.000,B 0.000,C 90.000,E1 140.275} C_DIS
LIN {X -0.126,Y -657.965,Z 1203.573,A 0.000,B 0.000,C 90.000,E1 139.057} C_DIS
LIN {X 0.227,Y -661.670,Z 1203.563,A 0.000,B 0.000,C 90.000,E1 137.310} C_DIS
LIN {X -0.301,Y -664.271,Z 1203.556,A 0.000,B 0.000,C 90.000,E1 136.134} C_DIS
LIN {X -0.317,Y -669.151,Z 1203.544,A 0.000,B 0.000,C 90.000,E1 133.947} C_DIS
LIN {X 0.234,Y -672.729,Z 1203.536,A 0.000,B 0.000,C 90.000,E1 132.447} C_DIS
LIN {X -0.041,Y -676.207,Z 1203.528,A 0.000,B 0.000,C 90.000,E1 131.024} C_DIS
LIN {X 0.195,Y -679.838,Z 1203.520,A 0.000,B 0.000,C 90.000,E1 129.564} C_DIS
LIN {X -0.374,Y -683.324,Z 1203.512,A 0.000,B 0.000,C 90.000,E1 128.177} C_DIS
LIN {X -0.299,Y -687.507,Z 1203.503,A 0.000,B 0.000,C 90.000,E1 126.503} C_DIS
LIN {X 0.142,Y -689.852,Z 1203.497,A 0.000,B 0.000,C 90.000,E1 125.518} C_DIS
LIN {X 0.117,Y -693.668,Z 1203.488,A 0.000,B 0.000,C 90.000,E1 123.865} C_DIS
LIN {X 0.288,Y -696.308,Z 1203.482,A 0.000,B 0.000,C 90.000,E1 122.673} C_DIS
LIN {X 0.363,Y -699.257,Z 1203.474,A 0.000,B 0.000,C 90.000,E1 121.258} C_DIS
LIN {X 0.136,Y -701.943,Z 1203.466,A 0.000,B 0.000,C 90.000,E1 119.873} C_DIS
LIN {X 0.295,Y -704.020,Z 1203.460,A 0.000,B 0.000,C 90.000,E1 118.693} C_DIS
LIN {X 0.195,Y -705.323,Z 1203.454,A 0.000,B 0.000,C 90.000,E1 117.769} C_DIS
LIN {X -0.222,Y -706.263,Z 1203.449,A 0.000,B 0.000,C 90.000,E1 116.873} C_DIS
LIN {X 0.009,Y -706.759,Z 1203.444,A 0.000,B 0.000,C 90.000,E1 115.924} C_DIS
LIN {X -0.332,Y -706.864,Z 1203.443,A 0.000,B 0.000,C 90.000,E1 115.720} C_DIS
LIN {X -0.094,Y -706.587,Z 1203.438,A 0.000,B 0.000,C 90.000,E1 114.771} C_DIS
LIN {X 0.199,Y -706.465,Z 1203.436,A 0.000,B 0.000,C 90.000,E1 114.515} C_DIS
LIN {X -0.152,Y -705.532,Z 1203.434,A 0.000,B 0.000,C 90.000,E1 114.079} C_DIS
LIN {X 0.137,Y -704.892,Z 1203.432,A 0.000,B 0.000,C 90.000,E1 113.823} C_DIS
LIN {X -0.220,Y -702.778,Z 1203.430,A 0.000,B 0.000,C 90.000,E1 113.387} C_DIS
LIN {X -0.081,Y -702.116,Z 1203.429,A 0.000,B 0.000,C 90.000,E1 113.259} C_DIS
LIN {X 0.057,Y -701.125,Z 1203.429,A 0.000,B 0.000,C 90.000,E1 113.131} C_DIS
LIN {X -0.002,Y -695.495,Z 1203.426,A 0.000,B 0.000,C 90.000,E1 112.695} C_DIS
LIN {X 0.065,Y -693.903,Z 1203.426,A 0.000,B 0.000,C 90.000,E1 112.589} C_DIS
LIN {X -0.241,Y -691.195,Z 1203.425,A 0.000,B 0.000,C 90.000,E1 112.514} C_DIS
LIN {X -0.032,Y -685.929,Z 1203.424,A 0.000,B 0.000,C 90.000,E1 112.333} C_DIS
LIN {X -0.343,Y -684.163,Z 1203.424,A 0.000,B 0.000,C 90.000,E1 112.333} C_DIS
LIN {X 0.017,Y -676.912,Z 1203.424,A 0.000,B 0.000,C 90.000,E1 112.280} C_DIS
LIN {X -0.032,Y -608.964,Z 1203.424,A 0.000,B 0.000,C 90.000,E1 112.280} C_DIS
LIN {X 0.162,Y -605.985,Z 1203.423,A 0.000,B 0.000,C 90.000,E1 112.078} C_DIS
LIN {X 0.087,Y -603.212,Z 1203.422,A 0.000,B 0.000,C 90.000,E1 111.897} C_DIS
LIN {X -0.136,Y -593.722,Z 1203.417,A 0.000,B 0.000,C 90.000,E1 111.153} C_DIS
LIN {X 0.096,Y -589.815,Z 1203.416,A 0.000,B 0.000,C 90.000,E1 110.791} C_DIS
LIN {X 0.252,Y -585.549,Z 1203.414,A 0.000,B 0.000,C 90.000,E1 110.429} C_DIS
LIN {X 0.130,Y -584.912,Z 1203.413,A 0.000,B 0.000,C 90.000,E1 110.375} C_DIS
LIN {X 0.093,Y -584.886,Z 1203.413,A 0.000,B 0.000,C 90.000,E1 110.375} C_DIS
LIN {X 0.157,Y -584.169,Z 1203.412,A 0.000,B 0.000,C 90.000,E1 110.120} C_DIS
LIN {X 0.101,Y -584.310,Z 1203.411,A 0.000,B 0.000,C 90.000,E1 109.993} C_DIS
LIN {X 0.168,Y -585.499,Z 1203.408,A 0.000,B 0.000,C 90.000,E1 109.450} C_DIS
LIN {X 0.006,Y -589.418,Z 1203.401,A 0.000,B 0.000,C 90.000,E1 108.127} C_DIS
LIN {X -0.090,Y -592.435,Z 1203.393,A 0.000,B 0.000,C 90.000,E1 106.804} C_DIS
LIN {X 0.032,Y -593.435,Z 1203.390,A 0.000,B 0.000,C 90.000,E1 106.260} C_DIS
LIN {X -0.143,Y -594.522,Z 1203.386,A 0.000,B 0.000,C 90.000,E1 105.481} C_DIS
LIN {X -0.169,Y -594.984,Z 1203.383,A 0.000,B 0.000,C 90.000,E1 104.954} C_DIS
LIN {X -0.038,Y -595.239,Z 1203.380,A 0.000,B 0.000,C 90.000,E1 104.411} C_DIS
LIN {X -0.056,Y -595.214,Z 1203.377,A 0.000,B 0.000,C 90.000,E1 103.883} C_DIS
LIN {X 0.226,Y -595.161,Z 1203.376,A 0.000,B 0.000,C 90.000,E1 103.592} C_DIS
LIN {X 0.213,Y -594.592,Z 1203.373,A 0.000,B 0.000,C 90.000,E1 103.063} C_DIS
LIN {X 0.197,Y -593.694,Z 1203.370,A 0.000,B 0.000,C 90.000,E1 102.535} C_DIS
LIN {X -0.102,Y -593.115,Z 1203.368,A 0.000,B 0.000,C 90.000,E1 102.299} C_DIS
LIN {X -0.127,Y -591.568,Z 1203.365,A 0.000,B 0.000,C 90.000,E1 101.771} C_DIS
LIN {X -0.163,Y -589.605,Z 1203.362,A 0.000,B 0.000,C 90.000,E1 101.243} C_DIS
LIN {X -0.214,Y -587.112,Z 1203.359,A 0.000,B 0.000,C 90.000,E1 100.715} C_DIS
LIN {X 0.184,Y -584.111,Z 1203.356,A 0.000,B 0.000,C 90.000,E1 100.141} C_DIS
LIN {X 0.308,Y -581.461,Z 1203.354,A 0.000,B 0.000,C 90.000,E1 99.726} C_DIS
LIN {X -0.253,Y -578.415,Z 1203.352,A 0.000,B 0.000,C 90.000,E1 99.378} C_DIS
LIN {X -0.249,Y -574.817,Z 1203.350,A 0.000,B 0.000,C 90.000,E1 98.973} C_DIS
LIN {X 0.152,Y -568.336,Z 1203.346,A 0.000,B 0.000,C 90.000,E1 98.276} C_DIS
LIN {X -0.216,Y -565.672,Z 1203.345,A 0.000,B 0.000,C 90.000,E1 98.049} C_DIS
LIN {X -0.187,Y -564.701,Z 1203.344,A 0.000,B 0.000,C 90.000,E1 97.936} C_DIS
LIN {X 0.066,Y -563.043,Z 1203.343,A 0.000,B 0.000,C 90.000,E1 97.644} C_DIS
LIN {X 0.104,Y -561.882,Z 1203.341,A 0.000,B 0.000,C 90.000,E1 97.296} C_DIS
LIN {X -0.107,Y -561.657,Z 1203.338,A 0.000,B 0.000,C 90.000,E1 96.834} C_DIS
LIN {X -0.025,Y -561.723,Z 1203.336,A 0.000,B 0.000,C 90.000,E1 96.549} C_DIS
LIN {X 0.120,Y -561.618,Z 1203.335,A 0.000,B 0.000,C 90.000,E1 96.258} C_DIS
LIN {X 0.006,Y -563.067,Z 1203.321,A 0.000,B 0.000,C 90.000,E1 93.784} C_DIS
LIN {X 0.085,Y -564.195,Z 1203.312,A 0.000,B 0.000,C 90.000,E1 92.121} C_DIS
LIN {X -0.262,Y -565.565,Z 1203.301,A 0.000,B 0.000,C 90.000,E1 90.229} C_DIS
LIN {X 0.194,Y -566.361,Z 1203.295,A 0.000,B 0.000,C 90.000,E1 89.083} C_DIS
LIN {X -0.223,Y -567.612,Z 1203.286,A 0.000,B 0.000,C 90.000,E1 87.478} C_DIS
LIN {X 0.104,Y -569.061,Z 1203.275,A 0.000,B 0.000,C 90.000,E1 85.527} C_DIS
LIN {X -0.174,Y -570.335,Z 1203.266,A 0.000,B 0.000,C 90.000,E1 83.913} C_DIS
LIN {X -0.239,Y -571.762,Z 1203.255,A 0.000,B 0.000,C 90.000,E1 82.008} C_DIS
LIN {X -0.022,Y -572.704,Z 1203.248,A 0.000,B 0.000,C 90.000,E1 80.622} C_DIS
LIN {X -0.163,Y -573.589,Z 1203.240,A 0.000,B 0.000,C 90.000,E1 79.275} C_DIS
LIN {X -0.189,Y -574.568,Z 1203.231,A 0.000,B 0.000,C 90.000,E1 77.645} C_DIS
LIN {X 0.046,Y -575.444,Z 1203.222,A 0.000,B 0.000,C 90.000,E1 75.992} C_DIS
LIN {X -0.053,Y -576.405,Z 1203.212,A 0.000,B 0.000,C 90.000,E1 74.102} C_DIS
LIN {X 0.167,Y -577.127,Z 1203.204,A 0.000,B 0.000,C 90.000,E1 72.725} C_DIS
LIN {X -0.151,Y -577.886,Z 1203.197,A 0.000,B 0.000,C 90.000,E1 71.402} C_DIS
LIN {X 0.142,Y -579.317,Z 1203.185,A 0.000,B 0.000,C 90.000,E1 69.209} C_DIS
LIN {X 0.144,Y -581.069,Z 1203.173,A 0.000,B 0.000,C 90.000,E1 67.050} C_DIS
LIN {X 0.015,Y -582.863,Z 1203.162,A 0.000,B 0.000,C 90.000,E1 65.177} C_DIS
LIN {X -0.098,Y -584.609,Z 1203.152,A 0.000,B 0.000,C 90.000,E1 63.307} C_DIS
LIN {X -0.190,Y -585.990,Z 1203.144,A 0.000,B 0.000,C 90.000,E1 61.975} C_DIS
LIN {X 0.050,Y -587.827,Z 1203.134,A 0.000,B 0.000,C 90.000,E1 60.078} C_DIS
LIN {X 0.054,Y -589.068,Z 1203.126,A 0.000,B 0.000,C 90.000,E1 58.742} C_DIS
LIN {X -0.224,Y -590.383,Z 1203.118,A 0.000,B 0.000,C 90.000,E1 57.168} C_DIS
LIN {X 0.143,Y -591.432,Z 1203.110,A 0.000,B 0.000,C 90.000,E1 55.801} C_DIS
LIN {X -0.365,Y -592.846,Z 1203.100,A 0.000,B 0.000,C 90.000,E1 53.989} C_DIS
LIN {X 0.285,Y -593.446,Z 1203.095,A 0.000,B 0.000,C 90.000,E1 53.130} C_DIS
LIN {X -0.140,Y -594.248,Z 1203.089,A 0.000,B 0.000,C 90.000,E1 52.110} C_DIS
LIN {X 0.110,Y -595.387,Z 1203.079,A 0.000,B 0.000,C 90.000,E1 50.231} C_DIS
LIN {X 0.083,Y -595.925,Z 1203.073,A 0.000,B 0.000,C 90.000,E1 49.175} C_DIS
LIN {X -0.166,Y -596.352,Z 1203.066,A 0.000,B 0.000,C 90.000,E1 47.877} C_DIS
LIN {X 0.218,Y -596.623,Z 1203.060,A 0.000,B 0.000,C 90.000,E1 46.782} C_DIS
LIN {X -0.045,Y -596.791,Z 1203.053,A 0.000,B 0.000,C 90.000,E1 45.486} C_DIS
LIN {X -0.079,Y -596.767,Z 1203.047,A 0.000,B 0.000,C 90.000,E1 44.433} C_DIS
LIN {X -0.120,Y -596.450,Z 1203.041,A 0.000,B 0.000,C 90.000,E1 43.380} C_DIS
LIN {X 0.039,Y -595.840,Z 1203.034,A 0.000,B 0.000,C 90.000,E1 42.043} C_DIS
LIN {X 0.015,Y -595.138,Z 1203.028,A 0.000,B 0.000,C 90.000,E1 40.987} C_DIS
LIN {X -0.016,Y -594.328,Z 1203.022,A 0.000,B 0.000,C 90.000,E1 39.930} C_DIS
LIN {X -0.062,Y -593.399,Z 1203.016,A 0.000,B 0.000,C 90.000,E1 38.874} C_DIS
LIN {X 0.187,Y -591.945,Z 1203.009,A 0.000,B 0.000,C 90.000,E1 37.523} C_DIS
LIN {X 0.000,Y -590.971,Z 1203.004,A 0.000,B 0.000,C 90.000,E1 36.744} C_DIS
LIN {X 0.014,Y -589.412,Z 1202.998,A 0.000,B 0.000,C 90.000,E1 35.678} C_DIS
LIN {X 0.195,Y -586.909,Z 1202.991,A 0.000,B 0.000,C 90.000,E1 34.326} C_DIS
LIN {X -0.376,Y -584.955,Z 1202.986,A 0.000,B 0.000,C 90.000,E1 33.579} C_DIS
LIN {X -0.153,Y -582.772,Z 1202.982,A 0.000,B 0.000,C 90.000,E1 32.752} C_DIS
LIN {X 0.042,Y -580.228,Z 1202.977,A 0.000,B 0.000,C 90.000,E1 31.926} C_DIS
LIN {X -0.097,Y -577.344,Z 1202.973,A 0.000,B 0.000,C 90.000,E1 31.131} C_DIS
LIN {X -0.260,Y -574.049,Z 1202.968,A 0.000,B 0.000,C 90.000,E1 30.335} C_DIS
LIN {X -0.212,Y -572.283,Z 1202.966,A 0.000,B 0.000,C 90.000,E1 29.922} C_DIS
LIN {X 0.059,Y -568.146,Z 1202.962,A 0.000,B 0.000,C 90.000,E1 29.077} C_DIS
LIN {X -0.116,Y -564.485,Z 1202.958,A 0.000,B 0.000,C 90.000,E1 28.409} C_DIS
LIN {X -0.094,Y -560.488,Z 1202.954,A 0.000,B 0.000,C 90.000,E1 27.719} C_DIS
LIN {X 0.049,Y -555.370,Z 1202.949,A 0.000,B 0.000,C 90.000,E1 26.873} C_DIS
LIN {X 0.001,Y -550.694,Z 1202.946,A 0.000,B 0.000,C 90.000,E1 26.181} C_DIS
LIN {X -0.104,Y -547.691,Z 1202.943,A 0.000,B 0.000,C 90.000,E1 25.771} C_DIS
LIN {X 0.144,Y -541.215,Z 1202.938,A 0.000,B 0.000,C 90.000,E1 24.899} C_DIS
LIN {X -0.024,Y -535.303,Z 1202.935,A 0.000,B 0.000,C 90.000,E1 24.207} C_DIS
LIN {X -0.231,Y -529.163,Z 1202.931,A 0.000,B 0.000,C 90.000,E1 23.515} C_DIS
LIN {X 0.069,Y -522.728,Z 1202.927,A 0.000,B 0.000,C 90.000,E1 22.770} C_DIS
LIN {X -0.007,Y -511.913,Z 1202.920,A 0.000,B 0.000,C 90.000,E1 21.663} C_DIS
LIN {X 0.077,Y -506.390,Z 1202.917,A 0.000,B 0.000,C 90.000,E1 21.099} C_DIS
LIN {X 0.091,Y -496.850,Z 1202.912,A 0.000,B 0.000,C 90.000,E1 20.174} C_DIS
LIN {X -0.175,Y -485.405,Z 1202.906,A 0.000,B 0.000,C 90.000,E1 19.141} C_DIS
LIN {X -0.110,Y -475.259,Z 1202.901,A 0.000,B 0.000,C 90.000,E1 18.236} C_DIS
LIN {X 0.023,Y -463.386,Z 1202.895,A 0.000,B 0.000,C 90.000,E1 17.166} C_DIS
LIN {X -0.091,Y -447.363,Z 1202.887,A 0.000,B 0.000,C 90.000,E1 15.717} C_DIS
LIN {X 0.096,Y -424.473,Z 1202.875,A 0.000,B 0.000,C 90.000,E1 13.411} C_DIS
LIN {X 0.163,Y -412.061,Z 1202.867,A 0.000,B 0.000,C 90.000,E1 12.007} C_DIS
LIN {X -0.154,Y -401.049,Z 1202.859,A 0.000,B 0.000,C 90.000,E1 10.715} C_DIS
LIN {X -0.151,Y -396.339,Z 1202.856,A 0.000,B 0.000,C 90.000,E1 10.018} C_DIS
LIN {X -0.070,Y -393.748,Z 1202.853,A 0.000,B 0.000,C 90.000,E1 9.500} C_DIS
LIN {X -0.075,Y -393.276,Z 1202.851,A 0.000,B 0.000,C 90.000,E1 9.208} C_DIS
LIN {X -0.113,Y -393.281,Z 1202.851,A 0.000,B 0.000,C 90.000,E1 9.208} C_DIS
LIN {X 0.094,Y -394.014,Z 1202.849,A 0.000,B 0.000,C 90.000,E1 8.746} C_DIS
LIN {X 0.021,Y -396.931,Z 1202.845,A 0.000,B 0.000,C 90.000,E1 8.049} C_DIS
LIN {X -0.221,Y -401.027,Z 1202.842,A 0.000,B 0.000,C 90.000,E1 7.530} C_DIS
LIN {X -0.027,Y -406.123,Z 1202.839,A 0.000,B 0.000,C 90.000,E1 6.947} C_DIS
LIN {X -0.108,Y -423.069,Z 1202.831,A 0.000,B 0.000,C 90.000,E1 5.625} C_DIS
LIN {X -0.083,Y -440.481,Z 1202.824,A 0.000,B 0.000,C 90.000,E1 4.302} C_DIS
LIN {X 0.084,Y -454.820,Z 1202.818,A 0.000,B 0.000,C 90.000,E1 3.212} C_DIS
LIN {X 0.049,Y -465.730,Z 1202.813,A 0.000,B 0.000,C 90.000,E1 2.407} C_DIS
LIN {X -0.153,Y -476.309,Z 1202.809,A 0.000,B 0.000,C 90.000,E1 1.604} C_DIS
LIN {X -0.091,Y -483.818,Z 1202.805,A 0.000,B 0.000,C 90.000,E1 0.974} C_DIS
LIN {X 0.230,Y -491.028,Z 1202.802,A 0.000,B 0.000,C 90.000,E1 0.286} C_DIS
LIN {X -0.011,Y -497.620,Z 1202.798,A 0.000,B 0.000,C 90.000,E1 359.656} C_DIS
LIN {X -0.254,Y -504.256,Z 1202.794,A 0.000,B 0.000,C 90.000,E1 358.969} C_DIS
LIN {X 0.051,Y -511.618,Z 1202.789,A 0.000,B 0.000,C 90.000,E1 358.051} C_DIS
LIN {X -0.117,Y -516.356,Z 1202.786,A 0.000,B 0.000,C 90.000,E1 357.478} C_DIS
LIN {X 0.002,Y -521.722,Z 1202.782,A 0.000,B 0.000,C 90.000,E1 356.731} C_DIS
LIN {X 0.137,Y -526.606,Z 1202.778,A 0.000,B 0.000,C 90.000,E1 355.988} C_DIS
LIN {X -0.176,Y -531.028,Z 1202.774,A 0.000,B 0.000,C 90.000,E1 355.298} C_DIS
LIN {X -0.179,Y -534.312,Z 1202.771,A 0.000,B 0.000,C 90.000,E1 354.723} C_DIS
LIN {X -0.157,Y -537.265,Z 1202.767,A 0.000,B 0.000,C 90.000,E1 354.147} C_DIS
LIN {X -0.252,Y -543.073,Z 1202.760,A 0.000,B 0.000,C 90.000,E1 352.875} C_DIS
LIN {X -0.085,Y -546.511,Z 1202.756,A 0.000,B 0.000,C 90.000,E1 352.008} C_DIS
LIN {X 0.119,Y -549.569,Z 1202.751,A 0.000,B 0.000,C 90.000,E1 351.141} C_DIS
LIN {X -0.192,Y -552.274,Z 1202.746,A 0.000,B 0.000,C 90.000,E1 350.330} C_DIS
LIN {X 0.164,Y -554.772,Z 1202.742,A 0.000,B 0.000,C 90.000,E1 349.454} C_DIS
LIN {X 0.144,Y -557.882,Z 1202.735,A 0.000,B 0.000,C 90.000,E1 348.342} C_DIS
LIN {X 0.022,Y -559.966,Z 1202.731,A 0.000,B 0.000,C 90.000,E1 347.521} C_DIS
LIN {X 0.072,Y -562.555,Z 1202.725,A 0.000,B 0.000,C 90.000,E1 346.408} C_DIS
LIN {X 0.289,Y -564.966,Z 1202.719,A 0.000,B 0.000,C 90.000,E1 345.283} C_DIS
LIN {X 0.163,Y -567.791,Z 1202.711,A 0.000,B 0.000,C 90.000,E1 343.921} C_DIS
LIN {X -0.137,Y -570.821,Z 1202.702,A 0.000,B 0.000,C 90.000,E1 342.308} C_DIS
LIN {X -0.190,Y -572.622,Z 1202.696,A 0.000,B 0.000,C 90.000,E1 341.221} C_DIS
LIN {X -0.024,Y -574.194,Z 1202.690,A 0.000,B 0.000,C 90.000,E1 340.115} C_DIS
LIN {X -0.033,Y -575.488,Z 1202.683,A 0.000,B 0.000,C 90.000,E1 339.028} C_DIS
LIN {X -0.199,Y -576.180,Z 1202.679,A 0.000,B 0.000,C 90.000,E1 338.230} C_DIS
LIN {X -0.141,Y -576.698,Z 1202.674,A 0.000,B 0.000,C 90.000,E1 337.411} C_DIS
LIN {X 0.080,Y -576.895,Z 1202.668,A 0.000,B 0.000,C 90.000,E1 336.305} C_DIS
LIN {X -0.222,Y -576.868,Z 1202.665,A 0.000,B 0.000,C 90.000,E1 335.793} C_DIS
LIN {X -0.147,Y -576.372,Z 1202.661,A 0.000,B 0.000,C 90.000,E1 334.973} C_DIS
LIN {X 0.074,Y -575.916,Z 1202.658,A 0.000,B 0.000,C 90.000,E1 334.409} C_DIS
LIN {X 0.134,Y -574.803,Z 1202.653,A 0.000,B 0.000,C 90.000,E1 333.589} C_DIS
LIN {X -0.072,Y -573.333,Z 1202.649,A 0.000,B 0.000,C 90.000,E1 332.794} C_DIS
LIN {X -0.044,Y -571.469,Z 1202.644,A 0.000,B 0.000,C 90.000,E1 331.975} C_DIS
LIN {X -0.273,Y -569.346,Z 1202.640,A 0.000,B 0.000,C 90.000,E1 331.179} C_DIS
LIN {X -0.024,Y -566.770,Z 1202.635,A 0.000,B 0.000,C 90.000,E1 330.333} C_DIS
LIN {X -0.297,Y -563.298,Z 1202.631,A 0.000,B 0.000,C 90.000,E1 329.537} C_DIS
LIN {X 0.078,Y -560.519,Z 1202.628,A 0.000,B 0.000,C 90.000,E1 328.948} C_DIS
LIN {X 0.056,Y -558.173,Z 1202.625,A 0.000,B 0.000,C 90.000,E1 328.535} C_DIS
LIN {X -0.087,Y -554.697,Z 1202.622,A 0.000,B 0.000,C 90.000,E1 327.995} C_DIS
LIN {X -0.075,Y -549.877,Z 1202.618,A 0.000,B 0.000,C 90.000,E1 327.296} C_DIS
LIN {X 0.224,Y -543.505,Z 1202.614,A 0.000,B 0.000,C 90.000,E1 326.421} C_DIS
LIN {X -0.005,Y -536.623,Z 1202.609,A 0.000,B 0.000,C 90.000,E1 325.595} C_DIS
LIN {X -0.221,Y -522.065,Z 1202.599,A 0.000,B 0.000,C 90.000,E1 323.909} C_DIS
LIN {X 0.108,Y -517.767,Z 1202.596,A 0.000,B 0.000,C 90.000,E1 323.290} C_DIS
LIN {X 0.022,Y -515.354,Z 1202.594,A 0.000,B 0.000,C 90.000,E1 322.924} C_DIS
LIN {X -0.180,Y -513.242,Z 1202.591,A 0.000,B 0.000,C 90.000,E1 322.477} C_DIS
LIN {X -0.059,Y -512.659,Z 1202.591,A 0.000,B 0.000,C 90.000,E1 322.316} C_DIS
LIN {X 0.004,Y -511.159,Z 1202.587,A 0.000,B 0.000,C 90.000,E1 321.698} C_DIS
LIN {X -0.049,Y -510.757,Z 1202.583,A 0.000,B 0.000,C 90.000,E1 320.964} C_DIS
LIN {X 0.180,Y -510.798,Z 1202.580,A 0.000,B 0.000,C 90.000,E1 320.356} C_DIS
LIN {X -0.015,Y -512.104,Z 1202.565,A 0.000,B 0.000,C 90.000,E1 317.715} C_DIS
LIN {X 0.183,Y -512.968,Z 1202.557,A 0.000,B 0.000,C 90.000,E1 316.215} C_DIS
LIN {X 0.296,Y -514.011,Z 1202.547,A 0.000,B 0.000,C 90.000,E1 314.433} C_DIS
LIN {X -0.193,Y -514.798,Z 1202.539,A 0.000,B 0.000,C 90.000,E1 313.014} C_DIS
LIN {X -0.021,Y -515.783,Z 1202.529,A 0.000,B 0.000,C 90.000,E1 311.229} C_DIS
LIN {X -0.106,Y -516.681,Z 1202.521,A 0.000,B 0.000,C 90.000,E1 309.769} C_DIS
LIN {X -0.049,Y -517.364,Z 1202.514,A 0.000,B 0.000,C 90.000,E1 308.588} C_DIS
LIN {X -0.301,Y -517.858,Z 1202.508,A 0.000,B 0.000,C 90.000,E1 307.443} C_DIS
LIN {X -0.355,Y -518.919,Z 1202.495,A 0.000,B 0.000,C 90.000,E1 305.105} C_DIS
LIN {X 0.212,Y -519.651,Z 1202.487,A 0.000,B 0.000,C 90.000,E1 303.579} C_DIS
LIN {X -0.270,Y -520.392,Z 1202.477,A 0.000,B 0.000,C 90.000,E1 301.878} C_DIS
LIN {X 0.098,Y -520.741,Z 1202.470,A 0.000,B 0.000,C 90.000,E1 300.669} C_DIS
LIN {X 0.084,Y -520.971,Z 1202.466,A 0.000,B 0.000,C 90.000,E1 299.795} C_DIS
LIN {X 0.249,Y -521.199,Z 1202.456,A 0.000,B 0.000,C 90.000,E1 298.025} C_DIS
LIN {X -0.061,Y -521.415,Z 1202.446,A 0.000,B 0.000,C 90.000,E1 296.309} C_DIS
LIN {X -0.184,Y -521.464,Z 1202.440,A 0.000,B 0.000,C 90.000,E1 295.155} C_DIS
LIN {X -0.166,Y -521.428,Z 1202.432,A 0.000,B 0.000,C 90.000,E1 293.695} C_DIS
LIN {X 0.267,Y -521.516,Z 1202.422,A 0.000,B 0.000,C 90.000,E1 291.897} C_DIS
LIN {X -0.129,Y -521.467,Z 1202.414,A 0.000,B 0.000,C 90.000,E1 290.482} C_DIS
LIN {X 0.149,Y -521.241,Z 1202.409,A 0.000,B 0.000,C 90.000,E1 289.577} C_DIS
LIN {X 0.065,Y -520.733,Z 1202.401,A 0.000,B 0.000,C 90.000,E1 288.127} C_DIS
LIN {X -0.033,Y -519.913,Z 1202.393,A 0.000,B 0.000,C 90.000,E1 286.677} C_DIS
LIN {X 0.200,Y -519.089,Z 1202.385,A 0.000,B 0.000,C 90.000,E1 285.190} C_DIS
LIN {X -0.104,Y -517.836,Z 1202.375,A 0.000,B 0.000,C 90.000,E1 283.467} C_DIS
LIN {X -0.183,Y -516.535,Z 1202.363,A 0.000,B 0.000,C 90.000,E1 281.422} C_DIS
LIN {X 0.236,Y -515.466,Z 1202.354,A 0.000,B 0.000,C 90.000,E1 279.613} C_DIS
LIN {X 0.076,Y -514.809,Z 1202.347,A 0.000,B 0.000,C 90.000,E1 278.454} C_DIS
LIN {X -0.125,Y -513.933,Z 1202.339,A 0.000,B 0.000,C 90.000,E1 277.004} C_DIS
LIN {X 0.007,Y -512.886,Z 1202.329,A 0.000,B 0.000,C 90.000,E1 275.220} C_DIS
LIN {X 0.166,Y -512.053,Z 1202.321,A 0.000,B 0.000,C 90.000,E1 273.726} C_DIS
LIN {X 0.041,Y -510.777,Z 1202.308,A 0.000,B 0.000,C 90.000,E1 271.375} C_DIS
LIN {X 0.119,Y -510.058,Z 1202.299,A 0.000,B 0.000,C 90.000,E1 269.885} C_DIS
LIN {X -0.235,Y -509.444,Z 1202.293,A 0.000,B 0.000,C 90.000,E1 268.740} C_DIS
LIN {X -0.077,Y -508.672,Z 1202.286,A 0.000,B 0.000,C 90.000,E1 267.535} C_DIS
LIN {X -0.029,Y -507.710,Z 1202.278,A 0.000,B 0.000,C 90.000,E1 266.045} C_DIS
LIN {X 0.137,Y -506.829,Z 1202.271,A 0.000,B 0.000,C 90.000,E1 264.837} C_DIS
LIN {X -0.097,Y -506.038,Z 1202.266,A 0.000,B 0.000,C 90.000,E1 263.970} C_DIS
LIN {X -0.141,Y -504.352,Z 1202.257,A 0.000,B 0.000,C 90.000,E1 262.186} C_DIS
LIN {X -0.156,Y -502.612,Z 1202.245,A 0.000,B 0.000,C 90.000,E1 260.095} C_DIS
LIN {X -0.192,Y -500.734,Z 1202.232,A 0.000,B 0.000,C 90.000,E1 257.701} C_DIS
LIN {X -0.069,Y -498.790,Z 1202.218,A 0.000,B 0.000,C 90.000,E1 255.283} C_DIS
LIN {X 0.112,Y -496.522,Z 1202.200,A 0.000,B 0.000,C 90.000,E1 251.945} C_DIS
LIN {X 0.141,Y -494.989,Z 1202.188,A 0.000,B 0.000,C 90.000,E1 249.826} C_DIS
LIN {X -0.125,Y -494.025,Z 1202.181,A 0.000,B 0.000,C 90.000,E1 248.646} C_DIS
LIN {X 0.017,Y -493.215,Z 1202.176,A 0.000,B 0.000,C 90.000,E1 247.720} C_DIS
LIN {X 0.148,Y -492.351,Z 1202.171,A 0.000,B 0.000,C 90.000,E1 246.794} C_DIS
LIN {X 0.087,Y -490.872,Z 1202.163,A 0.000,B 0.000,C 90.000,E1 245.281} C_DIS
LIN {X -0.004,Y -489.297,Z 1202.154,A 0.000,B 0.000,C 90.000,E1 243.768} C_DIS
LIN {X 0.083,Y -487.483,Z 1202.146,A 0.000,B 0.000,C 90.000,E1 242.231} C_DIS
LIN {X -0.064,Y -485.644,Z 1202.137,A 0.000,B 0.000,C 90.000,E1 240.717} C_DIS
LIN {X -0.018,Y -483.378,Z 1202.127,A 0.000,B 0.000,C 90.000,E1 238.869} C_DIS
LIN {X 0.001,Y -481.431,Z 1202.119,A 0.000,B 0.000,C 90.000,E1 237.327} C_DIS
LIN {X 0.041,Y -479.203,Z 1202.108,A 0.000,B 0.000,C 90.000,E1 235.468} C_DIS
LIN {X -0.084,Y -477.004,Z 1202.098,A 0.000,B 0.000,C 90.000,E1 233.623} C_DIS
LIN {X 0.279,Y -474.046,Z 1202.084,A 0.000,B 0.000,C 90.000,E1 231.090} C_DIS
LIN {X -0.054,Y -471.974,Z 1202.074,A 0.000,B 0.000,C 90.000,E1 229.256} C_DIS
LIN {X -0.096,Y -469.413,Z 1202.062,A 0.000,B 0.000,C 90.000,E1 227.067} C_DIS
LIN {X 0.270,Y -466.576,Z 1202.046,A 0.000,B 0.000,C 90.000,E1 224.190} C_DIS
LIN {X -0.095,Y -464.477,Z 1202.030,A 0.000,B 0.000,C 90.000,E1 221.391} C_DIS
LIN {X -0.134,Y -464.294,Z 1202.000,A 0.000,B 0.000,C 90.000,E1 216.011} C_DIS
LIN {X -0.063,Y -464.778,Z 1201.988,A 0.000,B 0.000,C 90.000,E1 213.785} C_DIS
LIN {X 0.063,Y -466.822,Z 1201.972,A 0.000,B 0.000,C 90.000,E1 210.924} C_DIS
LIN {X 0.185,Y -468.326,Z 1201.963,A 0.000,B 0.000,C 90.000,E1 209.333} C_DIS
LIN {X -0.262,Y -471.199,Z 1201.949,A 0.000,B 0.000,C 90.000,E1 206.873} C_DIS
LIN {X 0.086,Y -473.380,Z 1201.939,A 0.000,B 0.000,C 90.000,E1 204.951} C_DIS
LIN {X 0.022,Y -477.522,Z 1201.923,A 0.000,B 0.000,C 90.000,E1 202.153} C_DIS
LIN {X 0.220,Y -484.107,Z 1201.904,A 0.000,B 0.000,C 90.000,E1 198.725} C_DIS
LIN {X 0.098,Y -492.353,Z 1201.885,A 0.000,B 0.000,C 90.000,E1 195.371} C_DIS
LIN {X 0.141,Y -498.336,Z 1201.874,A 0.000,B 0.000,C 90.000,E1 193.244} C_DIS
LIN {X 0.230,Y -504.629,Z 1201.862,A 0.000,B 0.000,C 90.000,E1 191.130} C_DIS
LIN {X 0.222,Y -513.092,Z 1201.847,A 0.000,B 0.000,C 90.000,E1 188.454} C_DIS
LIN {X 0.035,Y -516.987,Z 1201.841,A 0.000,B 0.000,C 90.000,E1 187.296} C_DIS
LIN {X -0.175,Y -521.701,Z 1201.833,A 0.000,B 0.000,C 90.000,E1 185.853} C_DIS
LIN {X 0.172,Y -526.347,Z 1201.824,A 0.000,B 0.000,C 90.000,E1 184.359} C_DIS
LIN {X 0.059,Y -531.945,Z 1201.815,A 0.000,B 0.000,C 90.000,E1 182.636} C_DIS
LIN {X 0.045,Y -538.392,Z 1201.804,A 0.000,B 0.000,C 90.000,E1 180.630} C_DIS
LIN {X 0.131,Y -542.963,Z 1201.796,A 0.000,B 0.000,C 90.000,E1 179.198} C_DIS
LIN {X 0.272,Y -546.572,Z 1201.789,A 0.000,B 0.000,C 90.000,E1 178.051} C_DIS
LIN {X -0.025,Y -551.024,Z 1201.782,A 0.000,B 0.000,C 90.000,E1 176.674} C_DIS
LIN {X -0.257,Y -555.316,Z 1201.774,A 0.000,B 0.000,C 90.000,E1 175.298} C_DIS
LIN {X 0.234,Y -559.616,Z 1201.766,A 0.000,B 0.000,C 90.000,E1 173.856} C_DIS
LIN {X -0.064,Y -565.405,Z 1201.755,A 0.000,B 0.000,C 90.000,E1 171.951} C_DIS
LIN {X 0.227,Y -570.280,Z 1201.746,A 0.000,B 0.000,C 90.000,E1 170.274} C_DIS
LIN {X 0.058,Y -574.322,Z 1201.739,A 0.000,B 0.000,C 90.000,E1 168.926} C_DIS
LIN {X 0.061,Y -579.148,Z 1201.729,A 0.000,B 0.000,C 90.000,E1 167.297} C_DIS
LIN {X 0.181,Y -583.268,Z 1201.722,A 0.000,B 0.000,C 90.000,E1 165.936} C_DIS
LIN {X -0.262,Y -589.010,Z 1201.712,A 0.000,B 0.000,C 90.000,E1 164.102} C_DIS
LIN {X -0.241,Y -594.828,Z 1201.701,A 0.000,B 0.000,C 90.000,E1 162.236} C_DIS
LIN {X -0.242,Y -599.093,Z 1201.694,A 0.000,B 0.000,C 90.000,E1 160.913} C_DIS
LIN {X 0.220,Y -605.050,Z 1201.684,A 0.000,B 0.000,C 90.000,E1 159.028} C_DIS
LIN {X -0.036,Y -610.277,Z 1201.675,A 0.000,B 0.000,C 90.000,E1 157.486} C_DIS
LIN {X 0.081,Y -614.523,Z 1201.668,A 0.000,B 0.000,C 90.000,E1 156.177} C_DIS
LIN {X -0.294,Y -618.713,Z 1201.661,A 0.000,B 0.000,C 90.000,E1 154.921} C_DIS
LIN {X -0.337,Y -622.636,Z 1201.653,A 0.000,B 0.000,C 90.000,E1 153.640} C_DIS
LIN {X -0.299,Y -627.254,Z 1201.645,A 0.000,B 0.000,C 90.000,E1 152.103} C_DIS
LIN {X 0.073,Y -630.187,Z 1201.639,A 0.000,B 0.000,C 90.000,E1 151.051} C_DIS
LIN {X -0.026,Y -633.777,Z 1201.632,A 0.000,B 0.000,C 90.000,E1 149.793} C_DIS
LIN {X -0.068,Y -637.272,Z 1201.625,A 0.000,B 0.000,C 90.000,E1 148.535} C_DIS
LIN {X -0.109,Y -639.852,Z 1201.620,A 0.000,B 0.000,C 90.000,E1 147.533} C_DIS
